SPLINE
SPL {X  -157.404, Y  +360.095, Z    +0.000, E1   +17.695, E3 +109849.442}
SPL {X  -159.413, Y  +375.108, Z    +0.000, E1    +9.284, E3 +109858.530}
SPL {X  -159.978, Y  +386.135, Z    +0.000, E1    +2.544, E3 +109862.092}
SPL {X  -160.000, Y  +393.708, Z    +0.000, E1    -3.216, E3 +109863.846}
SPL {X  -160.000, Y  +400.474, Z    +0.000, E1    -9.529, E3 +109865.892}
SPL {X  -160.000, Y  +409.652, Z    +0.000, E1   -18.026, E3 +109870.028}
SPL {X  -160.000, Y  +437.804, Z    +0.000, E1   -34.779, E3 +109894.821}
SPL {X  -160.000, Y  +463.067, Z    +0.000, E1   -38.672, E3 +109940.521}
SPL {X  -160.000, Y  +469.167, Z    +0.000, E1   -38.717, E3 +109956.627}
SPL {X  -160.000, Y  +476.691, Z    +0.000, E1   -38.728, E3 +109976.559}
SPL {X  -160.000, Y  +483.419, Z    +0.000, E1   -38.692, E3 +109994.459}
SPL {X  -160.000, Y  +489.013, Z    +0.000, E1   -38.683, E3 +110009.298}
SPL {X  -160.000, Y  +494.786, Z    +0.000, E1   -38.693, E3 +110024.608}
SPL {X  -160.000, Y  +500.108, Z    +0.000, E1   -38.668, E3 +110038.759}
SPL {X  -160.000, Y  +504.903, Z    +0.000, E1   -38.673, E3 +110051.480}
SPL {X  -160.000, Y  +510.180, Z    +0.000, E1   -38.675, E3 +110065.485}
SPL {X  -160.000, Y  +515.083, Z    +0.000, E1   -38.662, E3 +110078.505}
SPL {X  -160.000, Y  +520.479, Z    +0.000, E1   -38.692, E3 +110092.779}
SPL {X  -160.000, Y  +525.998, Z    +0.000, E1   -38.666, E3 +110107.457}
SPL {X  -160.000, Y  +531.341, Z    +0.000, E1   -38.684, E3 +110121.601}
SPL {X  -160.000, Y  +537.313, Z    +0.000, E1   -38.686, E3 +110137.441}
SPL {X  -160.000, Y  +543.203, Z    +0.000, E1   -38.679, E3 +110153.067}
SPL {X  -160.000, Y  +551.201, Z    +0.000, E1   -38.768, E3 +110174.128}
SPL {X  -160.000, Y  +561.335, Z    +0.000, E1   -38.777, E3 +110200.998}
SPL {X  -160.000, Y  +568.812, Z    +0.000, E1   -38.671, E3 +110221.001}
SPL {X  -160.000, Y  +574.116, Z    +0.000, E1   -38.680, E3 +110235.072}
SPL {X  -160.000, Y  +582.193, Z    +0.000, E1   -38.759, E3 +110256.375}
SPL {X  -160.000, Y  +591.932, Z    +0.000, E1   -38.763, E3 +110282.200}
SPL {X  -160.000, Y  +601.488, Z    +0.000, E1   -38.747, E3 +110307.576}
SPL {X  -160.000, Y  +609.161, Z    +0.000, E1   -38.685, E3 +110328.027}
SPL {X  -160.000, Y  +614.445, Z    +0.000, E1   -38.661, E3 +110342.077}
SPL {X  -160.000, Y  +621.895, Z    +0.000, E1   -38.769, E3 +110361.665}
SPL {X  -160.000, Y  +631.692, Z    +0.000, E1   -38.748, E3 +110387.718}
SPL {X  -160.000, Y  +639.246, Z    +0.000, E1   -38.671, E3 +110407.894}
SPL {X  -160.000, Y  +644.827, Z    +0.000, E1   -38.662, E3 +110422.728}
SPL {X  -160.000, Y  +650.491, Z    +0.000, E1   -38.673, E3 +110437.716}
SPL {X  -160.000, Y  +656.011, Z    +0.000, E1   -38.669, E3 +110452.369}
SPL {X  -160.000, Y  +661.156, Z    +0.000, E1   -38.659, E3 +110466.044}
SPL {X  -160.000, Y  +666.701, Z    +0.000, E1   -38.683, E3 +110480.704}
SPL {X  -159.961, Y  +675.011, Z    +0.000, E1   -38.755, E3 +110502.691}
SPL {X  -159.451, Y  +684.743, Z    +0.000, E1   -38.666, E3 +110529.044}
SPL {X  -158.386, Y  +694.170, Z    +0.000, E1   -38.484, E3 +110555.163}
SPL {X  -157.286, Y  +700.846, Z    +0.000, E1   -38.194, E3 +110574.130}
SPL {X  -156.328, Y  +705.580, Z    +0.000, E1   -38.037, E3 +110587.666}
SPL {X  -155.162, Y  +710.549, Z    +0.000, E1   -37.822, E3 +110602.070}
SPL {X  -153.914, Y  +715.210, Z    +0.000, E1   -37.596, E3 +110615.720}
SPL {X  -152.686, Y  +719.322, Z    +0.000, E1   -37.361, E3 +110627.892}
SPL {X  -150.251, Y  +726.496, Z    +0.000, E1   -33.848, E3 +110676.388}
ENDSPLINE

SPLINE
SPL {X  -156.089, Y  +706.662, Z    +0.000, E1   -21.279, E3 +110729.041}
SPL {X  -159.059, Y  +688.824, Z    +0.000, E1   -11.551, E3 +110743.002}
SPL {X  -159.959, Y  +675.119, Z    +0.000, E1    -3.373, E3 +110747.830}
SPL {X  -160.000, Y  +666.447, Z    +0.000, E1    +3.005, E3 +110749.864}
SPL {X  -160.000, Y  +658.774, Z    +0.000, E1   +10.317, E3 +110752.123}
SPL {X  -160.000, Y  +647.765, Z    +0.000, E1   +20.359, E3 +110757.488}
SPL {X  -160.000, Y  +622.607, Z    +0.000, E1   +34.692, E3 +110780.356}
SPL {X  -160.000, Y  +596.106, Z    +0.000, E1   +39.718, E3 +110822.356}
SPL {X  -160.000, Y  +592.273, Z    +0.000, E1   +39.746, E3 +110832.093}
SPL {X  -160.000, Y  +586.287, Z    +0.000, E1   +39.762, E3 +110847.352}
SPL {X  -160.000, Y  +577.753, Z    +0.000, E1   +39.844, E3 +110868.994}
SPL {X  -160.000, Y  +567.367, Z    +0.000, E1   +39.853, E3 +110895.488}
SPL {X  -160.000, Y  +559.466, Z    +0.000, E1   +39.761, E3 +110915.770}
SPL {X  -160.000, Y  +552.914, Z    +0.000, E1   +39.787, E3 +110932.437}
SPL {X  -160.000, Y  +546.390, Z    +0.000, E1   +39.760, E3 +110949.151}
SPL {X  -160.000, Y  +540.123, Z    +0.000, E1   +39.770, E3 +110965.130}
SPL {X  -160.000, Y  +533.658, Z    +0.000, E1   +39.771, E3 +110981.628}
SPL {X  -160.000, Y  +527.046, Z    +0.000, E1   +39.771, E3 +110998.504}
SPL {X  -160.000, Y  +521.063, Z    +0.000, E1   +39.756, E3 +111013.789}
SPL {X  -160.000, Y  +515.110, Z    +0.000, E1   +39.770, E3 +111028.961}
SPL {X  -160.000, Y  +508.717, Z    +0.000, E1   +39.766, E3 +111045.280}
SPL {X  -160.000, Y  +502.133, Z    +0.000, E1   +39.780, E3 +111062.046}
ENDSPLINE

SPLINE
SPL {X  -160.000, Y  +512.949, Z    +0.000, E1   +32.050, E3 +111078.304}
ENDSPLINE

SPLINE
SPL {X  -160.000, Y  +507.092, Z    +0.000, E1   +32.805, E3 +111092.932}
SPL {X  -160.000, Y  +499.824, Z    +0.000, E1   +34.003, E3 +111108.674}
SPL {X  -160.000, Y  +491.367, Z    +0.000, E1   +35.449, E3 +111125.414}
SPL {X  -160.000, Y  +483.082, Z    +0.000, E1   +36.782, E3 +111141.253}
SPL {X  -160.000, Y  +474.521, Z    +0.000, E1   +38.037, E3 +111157.341}
SPL {X  -160.000, Y  +465.343, Z    +0.000, E1   +38.802, E3 +111177.500}
SPL {X  -160.000, Y  +457.266, Z    +0.000, E1   +38.756, E3 +111198.953}
SPL {X  -160.000, Y  +448.553, Z    +0.000, E1   +38.823, E3 +111221.904}
SPL {X  -160.000, Y  +439.425, Z    +0.000, E1   +38.797, E3 +111246.075}
SPL {X  -160.000, Y  +430.351, Z    +0.000, E1   +38.810, E3 +111270.090}
SPL {X  -160.000, Y  +421.477, Z    +0.000, E1   +38.792, E3 +111293.594}
SPL {X  -160.000, Y  +412.292, Z    +0.000, E1   +38.825, E3 +111317.821}
SPL {X  -160.000, Y  +403.281, Z    +0.000, E1   +38.797, E3 +111341.701}
SPL {X  -160.000, Y  +394.948, Z    +0.000, E1   +38.796, E3 +111363.743}
SPL {X  -159.971, Y  +385.741, Z    +0.000, E1   +38.831, E3 +111388.064}
SPL {X  -159.525, Y  +376.478, Z    +0.000, E1   +38.739, E3 +111413.055}
SPL {X  -158.721, Y  +368.613, Z    +0.000, E1   +38.561, E3 +111434.778}
SPL {X  -157.505, Y  +360.654, Z    +0.000, E1   +38.390, E3 +111457.052}
SPL {X  -156.229, Y  +354.269, Z    +0.000, E1   +38.076, E3 +111475.401}
SPL {X  -155.202, Y  +349.910, Z    +0.000, E1   +37.893, E3 +111487.976}
SPL {X  -154.128, Y  +345.852, Z    +0.000, E1   +37.701, E3 +111499.800}
SPL {X  -152.890, Y  +341.633, Z    +0.000, E1   +37.487, E3 +111512.232}
SPL {X  -150.284, Y  +333.893, Z    +0.000, E1   +33.433, E3 +111567.042}
ENDSPLINE

SPLINE
SPL {X  -157.404, Y  +360.095, Z    +0.000, E1   +17.695, E3 +111622.167}
SPL {X  -159.413, Y  +375.108, Z    +0.000, E1    +9.284, E3 +111631.256}
SPL {X  -159.978, Y  +386.135, Z    +0.000, E1    +2.544, E3 +111634.817}
SPL {X  -160.000, Y  +393.708, Z    +0.000, E1    -3.216, E3 +111636.571}
SPL {X  -160.000, Y  +400.474, Z    +0.000, E1    -9.529, E3 +111638.617}
SPL {X  -160.000, Y  +409.652, Z    +0.000, E1   -18.026, E3 +111642.754}
SPL {X  -160.000, Y  +437.804, Z    +0.000, E1   -34.779, E3 +111667.546}
SPL {X  -160.000, Y  +463.067, Z    +0.000, E1   -38.672, E3 +111713.246}
SPL {X  -160.000, Y  +469.167, Z    +0.000, E1   -38.717, E3 +111729.353}
SPL {X  -160.000, Y  +476.691, Z    +0.000, E1   -38.728, E3 +111749.284}
SPL {X  -160.000, Y  +483.419, Z    +0.000, E1   -38.692, E3 +111767.185}
SPL {X  -160.000, Y  +489.013, Z    +0.000, E1   -38.683, E3 +111782.023}
SPL {X  -160.000, Y  +494.786, Z    +0.000, E1   -38.693, E3 +111797.333}
SPL {X  -160.000, Y  +500.108, Z    +0.000, E1   -38.668, E3 +111811.485}
SPL {X  -160.000, Y  +504.903, Z    +0.000, E1   -38.673, E3 +111824.206}
SPL {X  -160.000, Y  +510.180, Z    +0.000, E1   -38.675, E3 +111838.210}
SPL {X  -160.000, Y  +515.083, Z    +0.000, E1   -38.662, E3 +111851.230}
SPL {X  -160.000, Y  +520.479, Z    +0.000, E1   -38.692, E3 +111865.504}
SPL {X  -160.000, Y  +525.998, Z    +0.000, E1   -38.666, E3 +111880.182}
SPL {X  -160.000, Y  +531.341, Z    +0.000, E1   -38.684, E3 +111894.327}
SPL {X  -160.000, Y  +537.313, Z    +0.000, E1   -38.686, E3 +111910.166}
SPL {X  -160.000, Y  +543.203, Z    +0.000, E1   -38.679, E3 +111925.792}
SPL {X  -160.000, Y  +551.201, Z    +0.000, E1   -38.768, E3 +111946.853}
SPL {X  -160.000, Y  +561.335, Z    +0.000, E1   -38.777, E3 +111973.723}
SPL {X  -160.000, Y  +568.812, Z    +0.000, E1   -38.671, E3 +111993.727}
SPL {X  -160.000, Y  +574.116, Z    +0.000, E1   -38.680, E3 +112007.797}
SPL {X  -160.000, Y  +582.193, Z    +0.000, E1   -38.759, E3 +112029.101}
SPL {X  -160.000, Y  +591.932, Z    +0.000, E1   -38.763, E3 +112054.926}
SPL {X  -160.000, Y  +601.488, Z    +0.000, E1   -38.747, E3 +112080.301}
SPL {X  -160.000, Y  +609.161, Z    +0.000, E1   -38.685, E3 +112100.753}
SPL {X  -160.000, Y  +614.445, Z    +0.000, E1   -38.661, E3 +112114.802}
SPL {X  -160.000, Y  +621.895, Z    +0.000, E1   -38.769, E3 +112134.390}
SPL {X  -160.000, Y  +631.692, Z    +0.000, E1   -38.748, E3 +112160.443}
SPL {X  -160.000, Y  +639.246, Z    +0.000, E1   -38.671, E3 +112180.619}
SPL {X  -160.000, Y  +644.827, Z    +0.000, E1   -38.662, E3 +112195.454}
SPL {X  -160.000, Y  +650.491, Z    +0.000, E1   -38.673, E3 +112210.441}
SPL {X  -160.000, Y  +656.011, Z    +0.000, E1   -38.669, E3 +112225.094}
SPL {X  -160.000, Y  +661.156, Z    +0.000, E1   -38.659, E3 +112238.769}
SPL {X  -160.000, Y  +666.701, Z    +0.000, E1   -38.683, E3 +112253.429}
SPL {X  -159.961, Y  +675.011, Z    +0.000, E1   -38.755, E3 +112275.416}
SPL {X  -159.451, Y  +684.743, Z    +0.000, E1   -38.666, E3 +112301.769}
SPL {X  -158.386, Y  +694.170, Z    +0.000, E1   -38.484, E3 +112327.888}
SPL {X  -157.286, Y  +700.846, Z    +0.000, E1   -38.194, E3 +112346.856}
SPL {X  -156.328, Y  +705.580, Z    +0.000, E1   -38.037, E3 +112360.392}
SPL {X  -155.162, Y  +710.549, Z    +0.000, E1   -37.822, E3 +112374.796}
SPL {X  -153.914, Y  +715.210, Z    +0.000, E1   -37.596, E3 +112388.445}
SPL {X  -152.686, Y  +719.322, Z    +0.000, E1   -37.361, E3 +112400.617}
SPL {X  -150.251, Y  +726.496, Z    +0.000, E1   -33.848, E3 +112449.113}
ENDSPLINE

SPLINE
SPL {X  -156.089, Y  +706.662, Z    +0.000, E1   -21.279, E3 +112501.766}
SPL {X  -159.059, Y  +688.824, Z    +0.000, E1   -11.551, E3 +112515.727}
SPL {X  -159.959, Y  +675.119, Z    +0.000, E1    -3.373, E3 +112520.555}
SPL {X  -160.000, Y  +666.447, Z    +0.000, E1    +3.005, E3 +112522.590}
SPL {X  -160.000, Y  +658.774, Z    +0.000, E1   +10.317, E3 +112524.848}
SPL {X  -160.000, Y  +647.765, Z    +0.000, E1   +20.359, E3 +112530.213}
SPL {X  -160.000, Y  +622.607, Z    +0.000, E1   +34.692, E3 +112553.081}
SPL {X  -160.000, Y  +593.120, Z    +0.000, E1   +39.775, E3 +112602.611}
SPL {X  -160.000, Y  +586.287, Z    +0.000, E1   +39.762, E3 +112620.078}
SPL {X  -160.000, Y  +577.753, Z    +0.000, E1   +39.844, E3 +112641.719}
SPL {X  -160.000, Y  +567.367, Z    +0.000, E1   +39.853, E3 +112668.213}
SPL {X  -160.000, Y  +559.466, Z    +0.000, E1   +39.761, E3 +112688.495}
SPL {X  -160.000, Y  +552.914, Z    +0.000, E1   +39.787, E3 +112705.162}
SPL {X  -160.000, Y  +546.390, Z    +0.000, E1   +39.760, E3 +112721.876}
SPL {X  -160.000, Y  +540.123, Z    +0.000, E1   +39.770, E3 +112737.855}
SPL {X  -160.000, Y  +533.658, Z    +0.000, E1   +39.771, E3 +112754.354}
SPL {X  -160.000, Y  +527.046, Z    +0.000, E1   +39.771, E3 +112771.230}
SPL {X  -160.000, Y  +521.063, Z    +0.000, E1   +39.756, E3 +112786.514}
SPL {X  -160.000, Y  +515.110, Z    +0.000, E1   +39.770, E3 +112801.687}
SPL {X  -160.000, Y  +508.717, Z    +0.000, E1   +39.766, E3 +112818.005}
SPL {X  -160.000, Y  +502.133, Z    +0.000, E1   +39.780, E3 +112834.771}
ENDSPLINE

SPLINE
SPL {X  -160.000, Y  +512.949, Z    +0.000, E1   +32.050, E3 +112851.029}
ENDSPLINE

SPLINE
SPL {X  -160.000, Y  +507.092, Z    +0.000, E1   +32.805, E3 +112865.657}
SPL {X  -160.000, Y  +499.824, Z    +0.000, E1   +34.003, E3 +112881.399}
SPL {X  -160.000, Y  +491.367, Z    +0.000, E1   +35.449, E3 +112898.139}
SPL {X  -160.000, Y  +483.082, Z    +0.000, E1   +36.782, E3 +112913.978}
SPL {X  -160.000, Y  +474.521, Z    +0.000, E1   +38.037, E3 +112930.066}
SPL {X  -160.000, Y  +465.343, Z    +0.000, E1   +38.802, E3 +112950.225}
SPL {X  -160.000, Y  +457.266, Z    +0.000, E1   +38.756, E3 +112971.679}
SPL {X  -160.000, Y  +448.553, Z    +0.000, E1   +38.823, E3 +112994.630}
SPL {X  -160.000, Y  +439.425, Z    +0.000, E1   +38.797, E3 +113018.801}
SPL {X  -160.000, Y  +430.351, Z    +0.000, E1   +38.810, E3 +113042.815}
SPL {X  -160.000, Y  +421.477, Z    +0.000, E1   +38.792, E3 +113066.319}
SPL {X  -160.000, Y  +412.292, Z    +0.000, E1   +38.825, E3 +113090.547}
SPL {X  -160.000, Y  +403.281, Z    +0.000, E1   +38.797, E3 +113114.426}
SPL {X  -160.000, Y  +394.948, Z    +0.000, E1   +38.796, E3 +113136.468}
SPL {X  -159.971, Y  +385.741, Z    +0.000, E1   +38.831, E3 +113160.789}
SPL {X  -159.525, Y  +376.478, Z    +0.000, E1   +38.739, E3 +113185.780}
SPL {X  -158.721, Y  +368.613, Z    +0.000, E1   +38.561, E3 +113207.504}
SPL {X  -157.505, Y  +360.654, Z    +0.000, E1   +38.390, E3 +113229.777}
SPL {X  -156.229, Y  +354.269, Z    +0.000, E1   +38.076, E3 +113248.126}
SPL {X  -155.202, Y  +349.910, Z    +0.000, E1   +37.893, E3 +113260.701}
SPL {X  -154.128, Y  +345.852, Z    +0.000, E1   +37.701, E3 +113272.525}
SPL {X  -152.890, Y  +341.633, Z    +0.000, E1   +37.487, E3 +113284.957}
SPL {X  -150.284, Y  +333.893, Z    +0.000, E1   +33.433, E3 +113339.767}
ENDSPLINE

SPLINE
SPL {X  -157.404, Y  +360.095, Z    +0.000, E1   +17.695, E3 +113394.892}
SPL {X  -159.413, Y  +375.108, Z    +0.000, E1    +9.284, E3 +113403.981}
SPL {X  -159.978, Y  +386.135, Z    +0.000, E1    +2.544, E3 +113407.542}
SPL {X  -160.000, Y  +393.708, Z    +0.000, E1    -3.216, E3 +113409.296}
SPL {X  -160.000, Y  +400.474, Z    +0.000, E1    -9.529, E3 +113411.342}
SPL {X  -160.000, Y  +409.652, Z    +0.000, E1   -18.026, E3 +113415.479}
SPL {X  -160.000, Y  +437.804, Z    +0.000, E1   -34.779, E3 +113440.272}
SPL {X  -160.000, Y  +463.067, Z    +0.000, E1   -38.672, E3 +113485.972}
SPL {X  -160.000, Y  +469.167, Z    +0.000, E1   -38.717, E3 +113502.078}
SPL {X  -160.000, Y  +476.691, Z    +0.000, E1   -38.728, E3 +113522.009}
SPL {X  -160.000, Y  +483.419, Z    +0.000, E1   -38.692, E3 +113539.910}
SPL {X  -160.000, Y  +489.013, Z    +0.000, E1   -38.683, E3 +113554.748}
SPL {X  -160.000, Y  +494.786, Z    +0.000, E1   -38.693, E3 +113570.058}
SPL {X  -160.000, Y  +500.108, Z    +0.000, E1   -38.668, E3 +113584.210}
SPL {X  -160.000, Y  +504.903, Z    +0.000, E1   -38.673, E3 +113596.931}
SPL {X  -160.000, Y  +510.180, Z    +0.000, E1   -38.675, E3 +113610.935}
SPL {X  -160.000, Y  +515.083, Z    +0.000, E1   -38.662, E3 +113623.955}
SPL {X  -160.000, Y  +520.479, Z    +0.000, E1   -38.692, E3 +113638.229}
SPL {X  -160.000, Y  +525.998, Z    +0.000, E1   -38.666, E3 +113652.908}
SPL {X  -160.000, Y  +531.341, Z    +0.000, E1   -38.684, E3 +113667.052}
SPL {X  -160.000, Y  +537.313, Z    +0.000, E1   -38.686, E3 +113682.892}
SPL {X  -160.000, Y  +543.203, Z    +0.000, E1   -38.679, E3 +113698.517}
SPL {X  -160.000, Y  +551.201, Z    +0.000, E1   -38.768, E3 +113719.578}
SPL {X  -160.000, Y  +561.335, Z    +0.000, E1   -38.777, E3 +113746.449}
SPL {X  -160.000, Y  +568.812, Z    +0.000, E1   -38.671, E3 +113766.452}
SPL {X  -160.000, Y  +574.116, Z    +0.000, E1   -38.680, E3 +113780.522}
SPL {X  -160.000, Y  +582.193, Z    +0.000, E1   -38.759, E3 +113801.826}
SPL {X  -160.000, Y  +591.932, Z    +0.000, E1   -38.763, E3 +113827.651}
SPL {X  -160.000, Y  +601.488, Z    +0.000, E1   -38.747, E3 +113853.026}
SPL {X  -160.000, Y  +609.161, Z    +0.000, E1   -38.685, E3 +113873.478}
SPL {X  -160.000, Y  +614.445, Z    +0.000, E1   -38.661, E3 +113887.527}
SPL {X  -160.000, Y  +621.895, Z    +0.000, E1   -38.769, E3 +113907.115}
SPL {X  -160.000, Y  +631.692, Z    +0.000, E1   -38.748, E3 +113933.169}
SPL {X  -160.000, Y  +639.246, Z    +0.000, E1   -38.671, E3 +113953.344}
SPL {X  -160.000, Y  +644.827, Z    +0.000, E1   -38.662, E3 +113968.179}
SPL {X  -160.000, Y  +650.491, Z    +0.000, E1   -38.673, E3 +113983.166}
SPL {X  -160.000, Y  +656.011, Z    +0.000, E1   -38.669, E3 +113997.819}
SPL {X  -160.000, Y  +661.156, Z    +0.000, E1   -38.659, E3 +114011.494}
SPL {X  -160.000, Y  +666.701, Z    +0.000, E1   -38.683, E3 +114026.155}
SPL {X  -159.961, Y  +675.011, Z    +0.000, E1   -38.755, E3 +114048.141}
SPL {X  -159.451, Y  +684.743, Z    +0.000, E1   -38.666, E3 +114074.495}
SPL {X  -158.386, Y  +694.170, Z    +0.000, E1   -38.484, E3 +114100.613}
SPL {X  -157.286, Y  +700.846, Z    +0.000, E1   -38.194, E3 +114119.581}
SPL {X  -156.328, Y  +705.580, Z    +0.000, E1   -38.037, E3 +114133.117}
SPL {X  -155.162, Y  +710.549, Z    +0.000, E1   -37.822, E3 +114147.521}
SPL {X  -153.914, Y  +715.210, Z    +0.000, E1   -37.596, E3 +114161.170}
SPL {X  -152.686, Y  +719.322, Z    +0.000, E1   -37.361, E3 +114173.342}
SPL {X  -150.251, Y  +726.496, Z    +0.000, E1   -33.848, E3 +114221.838}
ENDSPLINE

SPLINE
SPL {X  -156.089, Y  +706.662, Z    +0.000, E1   -21.279, E3 +114274.491}
SPL {X  -159.059, Y  +688.824, Z    +0.000, E1   -11.551, E3 +114288.452}
SPL {X  -159.959, Y  +675.119, Z    +0.000, E1    -3.373, E3 +114293.280}
SPL {X  -160.000, Y  +666.447, Z    +0.000, E1    +3.005, E3 +114295.315}
SPL {X  -160.000, Y  +658.774, Z    +0.000, E1   +10.317, E3 +114297.574}
SPL {X  -160.000, Y  +647.765, Z    +0.000, E1   +20.359, E3 +114302.939}
SPL {X  -160.000, Y  +622.607, Z    +0.000, E1   +34.692, E3 +114325.806}
SPL {X  -160.000, Y  +596.106, Z    +0.000, E1   +39.718, E3 +114367.806}
SPL {X  -160.000, Y  +592.273, Z    +0.000, E1   +39.746, E3 +114377.543}
SPL {X  -160.000, Y  +586.287, Z    +0.000, E1   +39.762, E3 +114392.803}
SPL {X  -160.000, Y  +577.753, Z    +0.000, E1   +39.844, E3 +114414.444}
SPL {X  -160.000, Y  +567.367, Z    +0.000, E1   +39.853, E3 +114440.939}
SPL {X  -160.000, Y  +559.466, Z    +0.000, E1   +39.761, E3 +114461.220}
SPL {X  -160.000, Y  +552.914, Z    +0.000, E1   +39.787, E3 +114477.887}
SPL {X  -160.000, Y  +546.390, Z    +0.000, E1   +39.760, E3 +114494.601}
SPL {X  -160.000, Y  +540.123, Z    +0.000, E1   +39.770, E3 +114510.580}
SPL {X  -160.000, Y  +533.658, Z    +0.000, E1   +39.771, E3 +114527.079}
SPL {X  -160.000, Y  +527.046, Z    +0.000, E1   +39.771, E3 +114543.955}
SPL {X  -160.000, Y  +521.063, Z    +0.000, E1   +39.756, E3 +114559.239}
SPL {X  -160.000, Y  +515.110, Z    +0.000, E1   +39.770, E3 +114574.412}
SPL {X  -160.000, Y  +508.717, Z    +0.000, E1   +39.766, E3 +114590.730}
SPL {X  -160.000, Y  +502.133, Z    +0.000, E1   +39.780, E3 +114607.497}
ENDSPLINE

SPLINE
SPL {X  -160.000, Y  +512.949, Z    +0.000, E1   +32.050, E3 +114623.754}
ENDSPLINE

SPLINE
SPL {X  -160.000, Y  +507.092, Z    +0.000, E1   +32.805, E3 +114638.382}
SPL {X  -160.000, Y  +499.824, Z    +0.000, E1   +34.003, E3 +114654.124}
SPL {X  -160.000, Y  +491.367, Z    +0.000, E1   +35.449, E3 +114670.865}
SPL {X  -160.000, Y  +483.082, Z    +0.000, E1   +36.782, E3 +114686.703}
SPL {X  -160.000, Y  +474.521, Z    +0.000, E1   +38.037, E3 +114702.791}
SPL {X  -160.000, Y  +465.343, Z    +0.000, E1   +38.802, E3 +114722.950}
SPL {X  -160.000, Y  +457.266, Z    +0.000, E1   +38.756, E3 +114744.404}
SPL {X  -160.000, Y  +448.553, Z    +0.000, E1   +38.823, E3 +114767.355}
SPL {X  -160.000, Y  +439.425, Z    +0.000, E1   +38.797, E3 +114791.526}
SPL {X  -160.000, Y  +430.351, Z    +0.000, E1   +38.810, E3 +114815.541}
SPL {X  -160.000, Y  +421.477, Z    +0.000, E1   +38.792, E3 +114839.044}
SPL {X  -160.000, Y  +412.292, Z    +0.000, E1   +38.825, E3 +114863.272}
SPL {X  -160.000, Y  +403.281, Z    +0.000, E1   +38.797, E3 +114887.152}
SPL {X  -160.000, Y  +394.948, Z    +0.000, E1   +38.796, E3 +114909.193}
SPL {X  -159.971, Y  +385.741, Z    +0.000, E1   +38.831, E3 +114933.515}
SPL {X  -159.525, Y  +376.478, Z    +0.000, E1   +38.739, E3 +114958.506}
SPL {X  -158.721, Y  +368.613, Z    +0.000, E1   +38.561, E3 +114980.229}
SPL {X  -157.505, Y  +360.654, Z    +0.000, E1   +38.390, E3 +115002.502}
SPL {X  -156.229, Y  +354.269, Z    +0.000, E1   +38.076, E3 +115020.852}
SPL {X  -155.202, Y  +349.910, Z    +0.000, E1   +37.893, E3 +115033.426}
SPL {X  -154.128, Y  +345.852, Z    +0.000, E1   +37.701, E3 +115045.250}
SPL {X  -152.890, Y  +341.633, Z    +0.000, E1   +37.487, E3 +115057.682}
SPL {X  -150.284, Y  +333.893, Z    +0.000, E1   +33.433, E3 +115112.493}
ENDSPLINE

SPLINE
SPL {X  -157.404, Y  +360.095, Z    +0.000, E1   +17.695, E3 +115167.617}
SPL {X  -159.413, Y  +375.108, Z    +0.000, E1    +9.284, E3 +115176.706}
SPL {X  -159.978, Y  +386.135, Z    +0.000, E1    +2.544, E3 +115180.267}
SPL {X  -160.000, Y  +393.708, Z    +0.000, E1    -3.216, E3 +115182.021}
SPL {X  -160.000, Y  +400.474, Z    +0.000, E1    -9.529, E3 +115184.068}
SPL {X  -160.000, Y  +409.652, Z    +0.000, E1   -18.026, E3 +115188.204}
SPL {X  -160.000, Y  +437.804, Z    +0.000, E1   -34.779, E3 +115212.997}
SPL {X  -160.000, Y  +463.067, Z    +0.000, E1   -38.672, E3 +115258.697}
SPL {X  -160.000, Y  +469.167, Z    +0.000, E1   -38.717, E3 +115274.803}
SPL {X  -160.000, Y  +476.691, Z    +0.000, E1   -38.728, E3 +115294.735}
SPL {X  -160.000, Y  +483.419, Z    +0.000, E1   -38.692, E3 +115312.635}
SPL {X  -160.000, Y  +489.013, Z    +0.000, E1   -38.683, E3 +115327.474}
SPL {X  -160.000, Y  +494.786, Z    +0.000, E1   -38.693, E3 +115342.784}
SPL {X  -160.000, Y  +500.108, Z    +0.000, E1   -38.668, E3 +115356.935}
SPL {X  -160.000, Y  +504.903, Z    +0.000, E1   -38.673, E3 +115369.656}
SPL {X  -160.000, Y  +510.180, Z    +0.000, E1   -38.675, E3 +115383.661}
SPL {X  -160.000, Y  +515.083, Z    +0.000, E1   -38.662, E3 +115396.680}
SPL {X  -160.000, Y  +520.479, Z    +0.000, E1   -38.692, E3 +115410.955}
SPL {X  -160.000, Y  +525.998, Z    +0.000, E1   -38.666, E3 +115425.633}
SPL {X  -160.000, Y  +531.341, Z    +0.000, E1   -38.684, E3 +115439.777}
SPL {X  -160.000, Y  +537.313, Z    +0.000, E1   -38.686, E3 +115455.617}
SPL {X  -160.000, Y  +543.203, Z    +0.000, E1   -38.679, E3 +115471.242}
SPL {X  -160.000, Y  +551.201, Z    +0.000, E1   -38.768, E3 +115492.304}
SPL {X  -160.000, Y  +561.335, Z    +0.000, E1   -38.777, E3 +115519.174}
SPL {X  -160.000, Y  +568.812, Z    +0.000, E1   -38.671, E3 +115539.177}
SPL {X  -160.000, Y  +574.116, Z    +0.000, E1   -38.680, E3 +115553.248}
SPL {X  -160.000, Y  +582.193, Z    +0.000, E1   -38.759, E3 +115574.551}
SPL {X  -160.000, Y  +591.932, Z    +0.000, E1   -38.763, E3 +115600.376}
SPL {X  -160.000, Y  +601.488, Z    +0.000, E1   -38.747, E3 +115625.751}
SPL {X  -160.000, Y  +609.161, Z    +0.000, E1   -38.685, E3 +115646.203}
SPL {X  -160.000, Y  +614.445, Z    +0.000, E1   -38.661, E3 +115660.252}
SPL {X  -160.000, Y  +621.895, Z    +0.000, E1   -38.769, E3 +115679.840}
SPL {X  -160.000, Y  +631.692, Z    +0.000, E1   -38.748, E3 +115705.894}
SPL {X  -160.000, Y  +639.246, Z    +0.000, E1   -38.671, E3 +115726.069}
SPL {X  -160.000, Y  +644.827, Z    +0.000, E1   -38.662, E3 +115740.904}
SPL {X  -160.000, Y  +650.491, Z    +0.000, E1   -38.673, E3 +115755.892}
SPL {X  -160.000, Y  +656.011, Z    +0.000, E1   -38.669, E3 +115770.545}
SPL {X  -160.000, Y  +661.156, Z    +0.000, E1   -38.659, E3 +115784.220}
SPL {X  -160.000, Y  +666.701, Z    +0.000, E1   -38.683, E3 +115798.880}
SPL {X  -159.961, Y  +675.011, Z    +0.000, E1   -38.755, E3 +115820.866}
SPL {X  -159.451, Y  +684.743, Z    +0.000, E1   -38.666, E3 +115847.220}
SPL {X  -158.386, Y  +694.170, Z    +0.000, E1   -38.484, E3 +115873.338}
SPL {X  -157.286, Y  +700.846, Z    +0.000, E1   -38.194, E3 +115892.306}
SPL {X  -156.328, Y  +705.580, Z    +0.000, E1   -38.037, E3 +115905.842}
SPL {X  -155.162, Y  +710.549, Z    +0.000, E1   -37.822, E3 +115920.246}
SPL {X  -153.914, Y  +715.210, Z    +0.000, E1   -37.596, E3 +115933.895}
SPL {X  -152.686, Y  +719.322, Z    +0.000, E1   -37.361, E3 +115946.068}
SPL {X  -150.251, Y  +726.496, Z    +0.000, E1   -33.848, E3 +115994.563}
ENDSPLINE

SPLINE
SPL {X  -156.089, Y  +706.662, Z    +0.000, E1   -21.279, E3 +116047.217}
SPL {X  -159.059, Y  +688.824, Z    +0.000, E1   -11.551, E3 +116061.177}
SPL {X  -159.959, Y  +675.119, Z    +0.000, E1    -3.373, E3 +116066.005}
SPL {X  -160.000, Y  +666.447, Z    +0.000, E1    +3.005, E3 +116068.040}
SPL {X  -160.000, Y  +658.774, Z    +0.000, E1   +10.317, E3 +116070.299}
SPL {X  -160.000, Y  +647.765, Z    +0.000, E1   +20.359, E3 +116075.664}
SPL {X  -160.000, Y  +622.607, Z    +0.000, E1   +34.692, E3 +116098.531}
SPL {X  -160.000, Y  +593.120, Z    +0.000, E1   +39.775, E3 +116148.061}
SPL {X  -160.000, Y  +586.287, Z    +0.000, E1   +39.762, E3 +116165.528}
SPL {X  -160.000, Y  +577.753, Z    +0.000, E1   +39.844, E3 +116187.170}
SPL {X  -160.000, Y  +567.367, Z    +0.000, E1   +39.853, E3 +116213.664}
SPL {X  -160.000, Y  +559.466, Z    +0.000, E1   +39.761, E3 +116233.945}
SPL {X  -160.000, Y  +552.914, Z    +0.000, E1   +39.787, E3 +116250.613}
SPL {X  -160.000, Y  +546.390, Z    +0.000, E1   +39.760, E3 +116267.326}
SPL {X  -160.000, Y  +540.123, Z    +0.000, E1   +39.770, E3 +116283.306}
SPL {X  -160.000, Y  +533.658, Z    +0.000, E1   +39.771, E3 +116299.804}
SPL {X  -160.000, Y  +527.046, Z    +0.000, E1   +39.771, E3 +116316.680}
SPL {X  -160.000, Y  +521.063, Z    +0.000, E1   +39.756, E3 +116331.965}
SPL {X  -160.000, Y  +515.110, Z    +0.000, E1   +39.770, E3 +116347.137}
SPL {X  -160.000, Y  +508.717, Z    +0.000, E1   +39.766, E3 +116363.455}
SPL {X  -160.000, Y  +502.133, Z    +0.000, E1   +39.780, E3 +116380.222}
ENDSPLINE

SPLINE
SPL {X  -160.000, Y  +512.949, Z    +0.000, E1   +32.050, E3 +116396.479}
ENDSPLINE

SPLINE
SPL {X  -160.000, Y  +507.092, Z    +0.000, E1   +32.805, E3 +116411.108}
SPL {X  -160.000, Y  +499.824, Z    +0.000, E1   +34.003, E3 +116426.849}
SPL {X  -160.000, Y  +491.367, Z    +0.000, E1   +35.449, E3 +116443.590}
SPL {X  -160.000, Y  +483.082, Z    +0.000, E1   +36.782, E3 +116459.429}
SPL {X  -160.000, Y  +474.521, Z    +0.000, E1   +38.037, E3 +116475.517}
SPL {X  -160.000, Y  +465.343, Z    +0.000, E1   +38.802, E3 +116495.675}
SPL {X  -160.000, Y  +457.266, Z    +0.000, E1   +38.756, E3 +116517.129}
SPL {X  -160.000, Y  +448.553, Z    +0.000, E1   +38.823, E3 +116540.080}
SPL {X  -160.000, Y  +439.425, Z    +0.000, E1   +38.797, E3 +116564.251}
SPL {X  -160.000, Y  +430.351, Z    +0.000, E1   +38.810, E3 +116588.266}
SPL {X  -160.000, Y  +421.477, Z    +0.000, E1   +38.792, E3 +116611.770}
SPL {X  -160.000, Y  +412.292, Z    +0.000, E1   +38.825, E3 +116635.997}
SPL {X  -160.000, Y  +403.281, Z    +0.000, E1   +38.797, E3 +116659.877}
SPL {X  -160.000, Y  +394.948, Z    +0.000, E1   +38.796, E3 +116681.919}
SPL {X  -159.971, Y  +385.741, Z    +0.000, E1   +38.831, E3 +116706.240}
SPL {X  -159.525, Y  +376.478, Z    +0.000, E1   +38.739, E3 +116731.231}
SPL {X  -158.721, Y  +368.613, Z    +0.000, E1   +38.561, E3 +116752.954}
SPL {X  -157.505, Y  +360.654, Z    +0.000, E1   +38.390, E3 +116775.227}
SPL {X  -156.229, Y  +354.269, Z    +0.000, E1   +38.076, E3 +116793.577}
SPL {X  -155.202, Y  +349.910, Z    +0.000, E1   +37.893, E3 +116806.151}
SPL {X  -154.128, Y  +345.852, Z    +0.000, E1   +37.701, E3 +116817.975}
SPL {X  -152.890, Y  +341.633, Z    +0.000, E1   +37.487, E3 +116830.407}
SPL {X  -150.284, Y  +333.893, Z    +0.000, E1   +33.433, E3 +116885.218}
ENDSPLINE

SPLINE
SPL {X  -157.404, Y  +360.095, Z    +0.000, E1   +17.695, E3 +116940.343}
SPL {X  -159.413, Y  +375.108, Z    +0.000, E1    +9.284, E3 +116949.431}
SPL {X  -159.978, Y  +386.135, Z    +0.000, E1    +2.544, E3 +116952.993}
SPL {X  -160.000, Y  +393.708, Z    +0.000, E1    -3.216, E3 +116954.746}
SPL {X  -160.000, Y  +400.474, Z    +0.000, E1    -9.529, E3 +116956.793}
SPL {X  -160.000, Y  +409.652, Z    +0.000, E1   -18.026, E3 +116960.929}
SPL {X  -160.000, Y  +437.804, Z    +0.000, E1   -34.779, E3 +116985.722}
SPL {X  -160.000, Y  +463.067, Z    +0.000, E1   -38.672, E3 +117031.422}
SPL {X  -160.000, Y  +469.167, Z    +0.000, E1   -38.717, E3 +117047.528}
SPL {X  -160.000, Y  +476.691, Z    +0.000, E1   -38.728, E3 +117067.460}
SPL {X  -160.000, Y  +483.419, Z    +0.000, E1   -38.692, E3 +117085.360}
SPL {X  -160.000, Y  +489.013, Z    +0.000, E1   -38.683, E3 +117100.199}
SPL {X  -160.000, Y  +494.786, Z    +0.000, E1   -38.693, E3 +117115.509}
SPL {X  -160.000, Y  +500.108, Z    +0.000, E1   -38.668, E3 +117129.660}
SPL {X  -160.000, Y  +504.903, Z    +0.000, E1   -38.673, E3 +117142.381}
SPL {X  -160.000, Y  +510.180, Z    +0.000, E1   -38.675, E3 +117156.386}
SPL {X  -160.000, Y  +515.083, Z    +0.000, E1   -38.662, E3 +117169.405}
SPL {X  -160.000, Y  +520.479, Z    +0.000, E1   -38.692, E3 +117183.680}
SPL {X  -160.000, Y  +525.998, Z    +0.000, E1   -38.666, E3 +117198.358}
SPL {X  -160.000, Y  +531.341, Z    +0.000, E1   -38.684, E3 +117212.502}
SPL {X  -160.000, Y  +537.313, Z    +0.000, E1   -38.686, E3 +117228.342}
SPL {X  -160.000, Y  +543.203, Z    +0.000, E1   -38.679, E3 +117243.968}
SPL {X  -160.000, Y  +551.201, Z    +0.000, E1   -38.768, E3 +117265.029}
SPL {X  -160.000, Y  +561.335, Z    +0.000, E1   -38.777, E3 +117291.899}
SPL {X  -160.000, Y  +568.812, Z    +0.000, E1   -38.671, E3 +117311.902}
SPL {X  -160.000, Y  +574.116, Z    +0.000, E1   -38.680, E3 +117325.973}
SPL {X  -160.000, Y  +582.193, Z    +0.000, E1   -38.759, E3 +117347.276}
SPL {X  -160.000, Y  +591.932, Z    +0.000, E1   -38.763, E3 +117373.101}
SPL {X  -160.000, Y  +601.488, Z    +0.000, E1   -38.747, E3 +117398.477}
SPL {X  -160.000, Y  +609.161, Z    +0.000, E1   -38.685, E3 +117418.928}
SPL {X  -160.000, Y  +614.445, Z    +0.000, E1   -38.661, E3 +117432.978}
SPL {X  -160.000, Y  +621.895, Z    +0.000, E1   -38.769, E3 +117452.566}
SPL {X  -160.000, Y  +631.692, Z    +0.000, E1   -38.748, E3 +117478.619}
SPL {X  -160.000, Y  +639.246, Z    +0.000, E1   -38.671, E3 +117498.795}
SPL {X  -160.000, Y  +644.827, Z    +0.000, E1   -38.662, E3 +117513.629}
SPL {X  -160.000, Y  +650.491, Z    +0.000, E1   -38.673, E3 +117528.617}
SPL {X  -160.000, Y  +656.011, Z    +0.000, E1   -38.669, E3 +117543.270}
SPL {X  -160.000, Y  +661.156, Z    +0.000, E1   -38.659, E3 +117556.945}
SPL {X  -160.000, Y  +666.701, Z    +0.000, E1   -38.683, E3 +117571.605}
SPL {X  -159.961, Y  +675.011, Z    +0.000, E1   -38.755, E3 +117593.592}
SPL {X  -159.451, Y  +684.743, Z    +0.000, E1   -38.666, E3 +117619.945}
SPL {X  -158.386, Y  +694.170, Z    +0.000, E1   -38.484, E3 +117646.064}
SPL {X  -157.286, Y  +700.846, Z    +0.000, E1   -38.194, E3 +117665.031}
SPL {X  -156.328, Y  +705.580, Z    +0.000, E1   -38.037, E3 +117678.567}
SPL {X  -155.162, Y  +710.549, Z    +0.000, E1   -37.822, E3 +117692.971}
SPL {X  -153.914, Y  +715.210, Z    +0.000, E1   -37.596, E3 +117706.621}
SPL {X  -152.686, Y  +719.322, Z    +0.000, E1   -37.361, E3 +117718.793}
SPL {X  -150.251, Y  +726.496, Z    +0.000, E1   -33.848, E3 +117767.289}
ENDSPLINE

SPLINE
SPL {X  -156.089, Y  +706.662, Z    +0.000, E1   -21.279, E3 +117819.942}
SPL {X  -159.059, Y  +688.824, Z    +0.000, E1   -11.551, E3 +117833.902}
SPL {X  -159.959, Y  +675.119, Z    +0.000, E1    -3.373, E3 +117838.731}
SPL {X  -160.000, Y  +666.447, Z    +0.000, E1    +3.005, E3 +117840.765}
SPL {X  -160.000, Y  +658.774, Z    +0.000, E1   +10.317, E3 +117843.024}
SPL {X  -160.000, Y  +647.765, Z    +0.000, E1   +20.359, E3 +117848.389}
SPL {X  -160.000, Y  +622.607, Z    +0.000, E1   +34.692, E3 +117871.257}
SPL {X  -160.000, Y  +596.106, Z    +0.000, E1   +39.718, E3 +117913.256}
SPL {X  -160.000, Y  +592.273, Z    +0.000, E1   +39.746, E3 +117922.994}
SPL {X  -160.000, Y  +586.287, Z    +0.000, E1   +39.762, E3 +117938.253}
SPL {X  -160.000, Y  +577.753, Z    +0.000, E1   +39.844, E3 +117959.895}
SPL {X  -160.000, Y  +567.367, Z    +0.000, E1   +39.853, E3 +117986.389}
SPL {X  -160.000, Y  +559.466, Z    +0.000, E1   +39.761, E3 +118006.671}
SPL {X  -160.000, Y  +552.914, Z    +0.000, E1   +39.787, E3 +118023.338}
SPL {X  -160.000, Y  +546.390, Z    +0.000, E1   +39.760, E3 +118040.052}
SPL {X  -160.000, Y  +540.123, Z    +0.000, E1   +39.770, E3 +118056.031}
SPL {X  -160.000, Y  +533.658, Z    +0.000, E1   +39.771, E3 +118072.529}
SPL {X  -160.000, Y  +527.046, Z    +0.000, E1   +39.771, E3 +118089.405}
SPL {X  -160.000, Y  +521.063, Z    +0.000, E1   +39.756, E3 +118104.690}
SPL {X  -160.000, Y  +515.110, Z    +0.000, E1   +39.770, E3 +118119.862}
SPL {X  -160.000, Y  +508.717, Z    +0.000, E1   +39.766, E3 +118136.181}
SPL {X  -160.000, Y  +502.133, Z    +0.000, E1   +39.780, E3 +118152.947}
ENDSPLINE

SPLINE
SPL {X  -160.000, Y  +512.949, Z    +0.000, E1   +32.050, E3 +118169.204}
ENDSPLINE

SPLINE
SPL {X  -160.000, Y  +507.092, Z    +0.000, E1   +32.805, E3 +118183.833}
SPL {X  -160.000, Y  +499.824, Z    +0.000, E1   +34.003, E3 +118199.575}
SPL {X  -160.000, Y  +491.367, Z    +0.000, E1   +35.449, E3 +118216.315}
SPL {X  -160.000, Y  +483.082, Z    +0.000, E1   +36.782, E3 +118232.154}
SPL {X  -160.000, Y  +474.521, Z    +0.000, E1   +38.037, E3 +118248.242}
SPL {X  -160.000, Y  +465.343, Z    +0.000, E1   +38.802, E3 +118268.401}
SPL {X  -160.000, Y  +457.266, Z    +0.000, E1   +38.756, E3 +118289.854}
SPL {X  -160.000, Y  +448.553, Z    +0.000, E1   +38.823, E3 +118312.805}
SPL {X  -160.000, Y  +439.425, Z    +0.000, E1   +38.797, E3 +118336.976}
SPL {X  -160.000, Y  +430.351, Z    +0.000, E1   +38.810, E3 +118360.991}
SPL {X  -160.000, Y  +421.477, Z    +0.000, E1   +38.792, E3 +118384.495}
SPL {X  -160.000, Y  +412.292, Z    +0.000, E1   +38.825, E3 +118408.722}
SPL {X  -160.000, Y  +403.281, Z    +0.000, E1   +38.797, E3 +118432.602}
SPL {X  -160.000, Y  +394.948, Z    +0.000, E1   +38.796, E3 +118454.644}
SPL {X  -159.971, Y  +385.741, Z    +0.000, E1   +38.831, E3 +118478.965}
SPL {X  -159.525, Y  +376.478, Z    +0.000, E1   +38.739, E3 +118503.956}
SPL {X  -158.721, Y  +368.613, Z    +0.000, E1   +38.561, E3 +118525.679}
SPL {X  -157.505, Y  +360.654, Z    +0.000, E1   +38.390, E3 +118547.952}
SPL {X  -156.229, Y  +354.269, Z    +0.000, E1   +38.076, E3 +118566.302}
SPL {X  -155.202, Y  +349.910, Z    +0.000, E1   +37.893, E3 +118578.877}
SPL {X  -154.128, Y  +345.852, Z    +0.000, E1   +37.701, E3 +118590.701}
SPL {X  -152.890, Y  +341.633, Z    +0.000, E1   +37.487, E3 +118603.133}
SPL {X  -150.284, Y  +333.893, Z    +0.000, E1   +33.433, E3 +118657.943}
ENDSPLINE

SPLINE
SPL {X  -157.404, Y  +360.095, Z    +0.000, E1   +17.695, E3 +118713.068}
SPL {X  -159.413, Y  +375.108, Z    +0.000, E1    +9.284, E3 +118722.157}
SPL {X  -159.978, Y  +386.135, Z    +0.000, E1    +2.544, E3 +118725.718}
SPL {X  -160.000, Y  +393.708, Z    +0.000, E1    -3.216, E3 +118727.472}
SPL {X  -160.000, Y  +400.474, Z    +0.000, E1    -9.529, E3 +118729.518}
SPL {X  -160.000, Y  +409.652, Z    +0.000, E1   -18.026, E3 +118733.655}
SPL {X  -160.000, Y  +437.804, Z    +0.000, E1   -34.779, E3 +118758.447}
SPL {X  -160.000, Y  +463.067, Z    +0.000, E1   -38.672, E3 +118804.147}
SPL {X  -160.000, Y  +469.167, Z    +0.000, E1   -38.717, E3 +118820.254}
SPL {X  -160.000, Y  +476.691, Z    +0.000, E1   -38.728, E3 +118840.185}
SPL {X  -160.000, Y  +483.419, Z    +0.000, E1   -38.692, E3 +118858.085}
SPL {X  -160.000, Y  +489.013, Z    +0.000, E1   -38.683, E3 +118872.924}
SPL {X  -160.000, Y  +494.786, Z    +0.000, E1   -38.693, E3 +118888.234}
SPL {X  -160.000, Y  +500.108, Z    +0.000, E1   -38.668, E3 +118902.386}
SPL {X  -160.000, Y  +504.903, Z    +0.000, E1   -38.673, E3 +118915.107}
SPL {X  -160.000, Y  +510.180, Z    +0.000, E1   -38.675, E3 +118929.111}
SPL {X  -160.000, Y  +515.083, Z    +0.000, E1   -38.662, E3 +118942.131}
SPL {X  -160.000, Y  +520.479, Z    +0.000, E1   -38.692, E3 +118956.405}
SPL {X  -160.000, Y  +525.998, Z    +0.000, E1   -38.666, E3 +118971.083}
SPL {X  -160.000, Y  +531.341, Z    +0.000, E1   -38.684, E3 +118985.228}
SPL {X  -160.000, Y  +537.313, Z    +0.000, E1   -38.686, E3 +119001.067}
SPL {X  -160.000, Y  +543.203, Z    +0.000, E1   -38.679, E3 +119016.693}
SPL {X  -160.000, Y  +551.201, Z    +0.000, E1   -38.768, E3 +119037.754}
SPL {X  -160.000, Y  +561.335, Z    +0.000, E1   -38.777, E3 +119064.624}
SPL {X  -160.000, Y  +568.812, Z    +0.000, E1   -38.671, E3 +119084.628}
SPL {X  -160.000, Y  +574.116, Z    +0.000, E1   -38.680, E3 +119098.698}
SPL {X  -160.000, Y  +582.193, Z    +0.000, E1   -38.759, E3 +119120.002}
SPL {X  -160.000, Y  +591.932, Z    +0.000, E1   -38.763, E3 +119145.827}
SPL {X  -160.000, Y  +601.488, Z    +0.000, E1   -38.747, E3 +119171.202}
SPL {X  -160.000, Y  +609.161, Z    +0.000, E1   -38.685, E3 +119191.654}
SPL {X  -160.000, Y  +614.445, Z    +0.000, E1   -38.661, E3 +119205.703}
SPL {X  -160.000, Y  +621.895, Z    +0.000, E1   -38.769, E3 +119225.291}
SPL {X  -160.000, Y  +631.692, Z    +0.000, E1   -38.748, E3 +119251.344}
SPL {X  -160.000, Y  +639.246, Z    +0.000, E1   -38.671, E3 +119271.520}
SPL {X  -160.000, Y  +644.827, Z    +0.000, E1   -38.662, E3 +119286.355}
SPL {X  -160.000, Y  +650.491, Z    +0.000, E1   -38.673, E3 +119301.342}
SPL {X  -160.000, Y  +656.011, Z    +0.000, E1   -38.669, E3 +119315.995}
SPL {X  -160.000, Y  +661.156, Z    +0.000, E1   -38.659, E3 +119329.670}
SPL {X  -160.000, Y  +666.701, Z    +0.000, E1   -38.683, E3 +119344.330}
SPL {X  -159.961, Y  +675.011, Z    +0.000, E1   -38.755, E3 +119366.317}
SPL {X  -159.451, Y  +684.743, Z    +0.000, E1   -38.666, E3 +119392.670}
SPL {X  -158.386, Y  +694.170, Z    +0.000, E1   -38.484, E3 +119418.789}
SPL {X  -157.286, Y  +700.846, Z    +0.000, E1   -38.194, E3 +119437.757}
SPL {X  -156.328, Y  +705.580, Z    +0.000, E1   -38.037, E3 +119451.293}
SPL {X  -155.162, Y  +710.549, Z    +0.000, E1   -37.822, E3 +119465.696}
SPL {X  -153.914, Y  +715.210, Z    +0.000, E1   -37.596, E3 +119479.346}
SPL {X  -152.686, Y  +719.322, Z    +0.000, E1   -37.361, E3 +119491.518}
SPL {X  -150.251, Y  +726.496, Z    +0.000, E1   -33.848, E3 +119540.014}
ENDSPLINE

SPLINE
SPL {X  -156.089, Y  +706.662, Z    +0.000, E1   -21.279, E3 +119592.667}
SPL {X  -159.059, Y  +688.824, Z    +0.000, E1   -11.551, E3 +119606.628}
SPL {X  -159.959, Y  +675.119, Z    +0.000, E1    -3.373, E3 +119611.456}
SPL {X  -160.000, Y  +666.447, Z    +0.000, E1    +3.005, E3 +119613.491}
SPL {X  -160.000, Y  +658.774, Z    +0.000, E1   +10.317, E3 +119615.749}
SPL {X  -160.000, Y  +647.765, Z    +0.000, E1   +20.359, E3 +119621.114}
SPL {X  -160.000, Y  +622.607, Z    +0.000, E1   +34.692, E3 +119643.982}
SPL {X  -160.000, Y  +593.120, Z    +0.000, E1   +39.775, E3 +119693.512}
SPL {X  -160.000, Y  +586.287, Z    +0.000, E1   +39.762, E3 +119710.978}
SPL {X  -160.000, Y  +577.753, Z    +0.000, E1   +39.844, E3 +119732.620}
SPL {X  -160.000, Y  +567.367, Z    +0.000, E1   +39.853, E3 +119759.114}
SPL {X  -160.000, Y  +559.466, Z    +0.000, E1   +39.761, E3 +119779.396}
SPL {X  -160.000, Y  +552.914, Z    +0.000, E1   +39.787, E3 +119796.063}
SPL {X  -160.000, Y  +546.390, Z    +0.000, E1   +39.760, E3 +119812.777}
SPL {X  -160.000, Y  +540.123, Z    +0.000, E1   +39.770, E3 +119828.756}
SPL {X  -160.000, Y  +533.658, Z    +0.000, E1   +39.771, E3 +119845.255}
SPL {X  -160.000, Y  +527.046, Z    +0.000, E1   +39.771, E3 +119862.131}
SPL {X  -160.000, Y  +521.063, Z    +0.000, E1   +39.756, E3 +119877.415}
SPL {X  -160.000, Y  +515.110, Z    +0.000, E1   +39.770, E3 +119892.588}
SPL {X  -160.000, Y  +508.717, Z    +0.000, E1   +39.766, E3 +119908.906}
SPL {X  -160.000, Y  +502.133, Z    +0.000, E1   +39.780, E3 +119925.672}
ENDSPLINE

SPLINE
SPL {X  -160.000, Y  +512.949, Z    +0.000, E1   +32.050, E3 +119941.930}
ENDSPLINE

SPLINE
SPL {X  -160.000, Y  +507.092, Z    +0.000, E1   +32.805, E3 +119956.558}
SPL {X  -160.000, Y  +499.824, Z    +0.000, E1   +34.003, E3 +119972.300}
SPL {X  -160.000, Y  +491.367, Z    +0.000, E1   +35.449, E3 +119989.040}
SPL {X  -160.000, Y  +483.082, Z    +0.000, E1   +36.782, E3 +120004.879}
SPL {X  -160.000, Y  +474.521, Z    +0.000, E1   +38.037, E3 +120020.967}
SPL {X  -160.000, Y  +465.343, Z    +0.000, E1   +38.802, E3 +120041.126}
SPL {X  -160.000, Y  +457.266, Z    +0.000, E1   +38.756, E3 +120062.580}
SPL {X  -160.000, Y  +448.553, Z    +0.000, E1   +38.823, E3 +120085.531}
SPL {X  -160.000, Y  +439.425, Z    +0.000, E1   +38.797, E3 +120109.702}
SPL {X  -160.000, Y  +430.351, Z    +0.000, E1   +38.810, E3 +120133.716}
SPL {X  -160.000, Y  +421.477, Z    +0.000, E1   +38.792, E3 +120157.220}
SPL {X  -160.000, Y  +412.292, Z    +0.000, E1   +38.825, E3 +120181.447}
SPL {X  -160.000, Y  +403.281, Z    +0.000, E1   +38.797, E3 +120205.327}
SPL {X  -160.000, Y  +394.948, Z    +0.000, E1   +38.796, E3 +120227.369}
SPL {X  -159.971, Y  +385.741, Z    +0.000, E1   +38.831, E3 +120251.690}
SPL {X  -159.525, Y  +376.478, Z    +0.000, E1   +38.739, E3 +120276.681}
SPL {X  -158.721, Y  +368.613, Z    +0.000, E1   +38.561, E3 +120298.405}
SPL {X  -157.505, Y  +360.654, Z    +0.000, E1   +38.390, E3 +120320.678}
SPL {X  -156.229, Y  +354.269, Z    +0.000, E1   +38.076, E3 +120339.027}
SPL {X  -155.202, Y  +349.910, Z    +0.000, E1   +37.893, E3 +120351.602}
SPL {X  -154.128, Y  +345.852, Z    +0.000, E1   +37.701, E3 +120363.426}
SPL {X  -152.890, Y  +341.633, Z    +0.000, E1   +37.487, E3 +120375.858}
SPL {X  -150.284, Y  +333.893, Z    +0.000, E1   +33.433, E3 +120430.668}
ENDSPLINE

SPLINE
SPL {X  -157.404, Y  +360.095, Z    +0.000, E1   +17.695, E3 +120485.793}
SPL {X  -159.413, Y  +375.108, Z    +0.000, E1    +9.284, E3 +120494.882}
SPL {X  -159.978, Y  +386.135, Z    +0.000, E1    +2.544, E3 +120498.443}
SPL {X  -160.000, Y  +393.708, Z    +0.000, E1    -3.216, E3 +120500.197}
SPL {X  -160.000, Y  +400.474, Z    +0.000, E1    -9.529, E3 +120502.243}
SPL {X  -160.000, Y  +409.652, Z    +0.000, E1   -18.026, E3 +120506.380}
SPL {X  -160.000, Y  +437.804, Z    +0.000, E1   -34.779, E3 +120531.173}
SPL {X  -160.000, Y  +463.067, Z    +0.000, E1   -38.672, E3 +120576.873}
SPL {X  -160.000, Y  +469.167, Z    +0.000, E1   -38.717, E3 +120592.979}
SPL {X  -160.000, Y  +476.691, Z    +0.000, E1   -38.728, E3 +120612.910}
SPL {X  -160.000, Y  +483.419, Z    +0.000, E1   -38.692, E3 +120630.811}
SPL {X  -160.000, Y  +489.013, Z    +0.000, E1   -38.683, E3 +120645.649}
SPL {X  -160.000, Y  +494.786, Z    +0.000, E1   -38.693, E3 +120660.959}
SPL {X  -160.000, Y  +500.108, Z    +0.000, E1   -38.668, E3 +120675.111}
SPL {X  -160.000, Y  +504.903, Z    +0.000, E1   -38.673, E3 +120687.832}
SPL {X  -160.000, Y  +510.180, Z    +0.000, E1   -38.675, E3 +120701.836}
SPL {X  -160.000, Y  +515.083, Z    +0.000, E1   -38.662, E3 +120714.856}
SPL {X  -160.000, Y  +520.479, Z    +0.000, E1   -38.692, E3 +120729.130}
SPL {X  -160.000, Y  +525.998, Z    +0.000, E1   -38.666, E3 +120743.809}
SPL {X  -160.000, Y  +531.341, Z    +0.000, E1   -38.684, E3 +120757.953}
SPL {X  -160.000, Y  +537.313, Z    +0.000, E1   -38.686, E3 +120773.793}
SPL {X  -160.000, Y  +543.203, Z    +0.000, E1   -38.679, E3 +120789.418}
SPL {X  -160.000, Y  +551.201, Z    +0.000, E1   -38.768, E3 +120810.479}
SPL {X  -160.000, Y  +561.335, Z    +0.000, E1   -38.777, E3 +120837.350}
SPL {X  -160.000, Y  +568.812, Z    +0.000, E1   -38.671, E3 +120857.353}
SPL {X  -160.000, Y  +574.116, Z    +0.000, E1   -38.680, E3 +120871.423}
SPL {X  -160.000, Y  +582.193, Z    +0.000, E1   -38.759, E3 +120892.727}
SPL {X  -160.000, Y  +591.932, Z    +0.000, E1   -38.763, E3 +120918.552}
SPL {X  -160.000, Y  +601.488, Z    +0.000, E1   -38.747, E3 +120943.927}
SPL {X  -160.000, Y  +609.161, Z    +0.000, E1   -38.685, E3 +120964.379}
SPL {X  -160.000, Y  +614.445, Z    +0.000, E1   -38.661, E3 +120978.428}
SPL {X  -160.000, Y  +621.895, Z    +0.000, E1   -38.769, E3 +120998.016}
SPL {X  -160.000, Y  +631.692, Z    +0.000, E1   -38.748, E3 +121024.070}
SPL {X  -160.000, Y  +639.246, Z    +0.000, E1   -38.671, E3 +121044.245}
SPL {X  -160.000, Y  +644.827, Z    +0.000, E1   -38.662, E3 +121059.080}
SPL {X  -160.000, Y  +650.491, Z    +0.000, E1   -38.673, E3 +121074.067}
SPL {X  -160.000, Y  +656.011, Z    +0.000, E1   -38.669, E3 +121088.720}
SPL {X  -160.000, Y  +661.156, Z    +0.000, E1   -38.659, E3 +121102.395}
SPL {X  -160.000, Y  +666.701, Z    +0.000, E1   -38.683, E3 +121117.056}
SPL {X  -159.961, Y  +675.011, Z    +0.000, E1   -38.755, E3 +121139.042}
SPL {X  -159.451, Y  +684.743, Z    +0.000, E1   -38.666, E3 +121165.396}
SPL {X  -158.386, Y  +694.170, Z    +0.000, E1   -38.484, E3 +121191.514}
SPL {X  -157.286, Y  +700.846, Z    +0.000, E1   -38.194, E3 +121210.482}
SPL {X  -156.328, Y  +705.580, Z    +0.000, E1   -38.037, E3 +121224.018}
SPL {X  -155.162, Y  +710.549, Z    +0.000, E1   -37.822, E3 +121238.422}
SPL {X  -153.914, Y  +715.210, Z    +0.000, E1   -37.596, E3 +121252.071}
SPL {X  -152.686, Y  +719.322, Z    +0.000, E1   -37.361, E3 +121264.243}
SPL {X  -150.251, Y  +726.496, Z    +0.000, E1   -33.848, E3 +121312.739}
ENDSPLINE

SPLINE
SPL {X  -156.089, Y  +706.662, Z    +0.000, E1   -21.279, E3 +121365.392}
SPL {X  -159.059, Y  +688.824, Z    +0.000, E1   -11.551, E3 +121379.353}
SPL {X  -159.959, Y  +675.119, Z    +0.000, E1    -3.373, E3 +121384.181}
SPL {X  -160.000, Y  +666.447, Z    +0.000, E1    +3.005, E3 +121386.216}
SPL {X  -160.000, Y  +658.774, Z    +0.000, E1   +10.317, E3 +121388.474}
SPL {X  -160.000, Y  +647.765, Z    +0.000, E1   +20.359, E3 +121393.840}
SPL {X  -160.000, Y  +622.607, Z    +0.000, E1   +34.692, E3 +121416.707}
SPL {X  -160.000, Y  +596.106, Z    +0.000, E1   +39.718, E3 +121458.707}
SPL {X  -160.000, Y  +592.273, Z    +0.000, E1   +39.746, E3 +121468.444}
SPL {X  -160.000, Y  +586.287, Z    +0.000, E1   +39.762, E3 +121483.704}
SPL {X  -160.000, Y  +577.753, Z    +0.000, E1   +39.844, E3 +121505.345}
SPL {X  -160.000, Y  +567.367, Z    +0.000, E1   +39.853, E3 +121531.840}
SPL {X  -160.000, Y  +559.466, Z    +0.000, E1   +39.761, E3 +121552.121}
SPL {X  -160.000, Y  +552.914, Z    +0.000, E1   +39.787, E3 +121568.788}
SPL {X  -160.000, Y  +546.390, Z    +0.000, E1   +39.760, E3 +121585.502}
SPL {X  -160.000, Y  +540.123, Z    +0.000, E1   +39.770, E3 +121601.481}
SPL {X  -160.000, Y  +533.658, Z    +0.000, E1   +39.771, E3 +121617.980}
SPL {X  -160.000, Y  +527.046, Z    +0.000, E1   +39.771, E3 +121634.856}
SPL {X  -160.000, Y  +521.063, Z    +0.000, E1   +39.756, E3 +121650.140}
SPL {X  -160.000, Y  +515.110, Z    +0.000, E1   +39.770, E3 +121665.313}
SPL {X  -160.000, Y  +508.717, Z    +0.000, E1   +39.766, E3 +121681.631}
SPL {X  -160.000, Y  +502.133, Z    +0.000, E1   +39.780, E3 +121698.398}
ENDSPLINE

SPLINE
SPL {X  -160.000, Y  +512.949, Z    +0.000, E1   +32.050, E3 +121714.655}
ENDSPLINE

SPLINE
SPL {X  -160.000, Y  +507.092, Z    +0.000, E1   +32.805, E3 +121729.283}
SPL {X  -160.000, Y  +499.824, Z    +0.000, E1   +34.003, E3 +121745.025}
SPL {X  -160.000, Y  +491.367, Z    +0.000, E1   +35.449, E3 +121761.766}
SPL {X  -160.000, Y  +483.082, Z    +0.000, E1   +36.782, E3 +121777.604}
SPL {X  -160.000, Y  +474.521, Z    +0.000, E1   +38.037, E3 +121793.692}
SPL {X  -160.000, Y  +465.343, Z    +0.000, E1   +38.802, E3 +121813.851}
SPL {X  -160.000, Y  +457.266, Z    +0.000, E1   +38.756, E3 +121835.305}
SPL {X  -160.000, Y  +448.553, Z    +0.000, E1   +38.823, E3 +121858.256}
SPL {X  -160.000, Y  +439.425, Z    +0.000, E1   +38.797, E3 +121882.427}
SPL {X  -160.000, Y  +430.351, Z    +0.000, E1   +38.810, E3 +121906.442}
SPL {X  -160.000, Y  +421.477, Z    +0.000, E1   +38.792, E3 +121929.945}
SPL {X  -160.000, Y  +412.292, Z    +0.000, E1   +38.825, E3 +121954.173}
SPL {X  -160.000, Y  +403.281, Z    +0.000, E1   +38.797, E3 +121978.053}
SPL {X  -160.000, Y  +394.948, Z    +0.000, E1   +38.796, E3 +122000.094}
SPL {X  -159.971, Y  +385.741, Z    +0.000, E1   +38.831, E3 +122024.416}
SPL {X  -159.525, Y  +376.478, Z    +0.000, E1   +38.739, E3 +122049.407}
SPL {X  -158.721, Y  +368.613, Z    +0.000, E1   +38.561, E3 +122071.130}
SPL {X  -157.505, Y  +360.654, Z    +0.000, E1   +38.390, E3 +122093.403}
SPL {X  -156.229, Y  +354.269, Z    +0.000, E1   +38.076, E3 +122111.753}
SPL {X  -155.202, Y  +349.910, Z    +0.000, E1   +37.893, E3 +122124.327}
SPL {X  -154.128, Y  +345.852, Z    +0.000, E1   +37.701, E3 +122136.151}
SPL {X  -152.890, Y  +341.633, Z    +0.000, E1   +37.487, E3 +122148.583}
SPL {X  -150.284, Y  +333.893, Z    +0.000, E1   +33.433, E3 +122203.394}
ENDSPLINE

SPLINE
SPL {X  -157.404, Y  +360.095, Z    +0.000, E1   +17.695, E3 +122258.518}
SPL {X  -159.413, Y  +375.108, Z    +0.000, E1    +9.284, E3 +122267.607}
SPL {X  -159.978, Y  +386.135, Z    +0.000, E1    +2.544, E3 +122271.168}
SPL {X  -160.000, Y  +393.708, Z    +0.000, E1    -3.216, E3 +122272.922}
SPL {X  -160.000, Y  +400.474, Z    +0.000, E1    -9.529, E3 +122274.969}
SPL {X  -160.000, Y  +409.652, Z    +0.000, E1   -18.026, E3 +122279.105}
SPL {X  -160.000, Y  +437.804, Z    +0.000, E1   -34.779, E3 +122303.898}
SPL {X  -160.000, Y  +463.067, Z    +0.000, E1   -38.672, E3 +122349.598}
SPL {X  -160.000, Y  +469.167, Z    +0.000, E1   -38.717, E3 +122365.704}
SPL {X  -160.000, Y  +476.691, Z    +0.000, E1   -38.728, E3 +122385.636}
SPL {X  -160.000, Y  +483.419, Z    +0.000, E1   -38.692, E3 +122403.536}
SPL {X  -160.000, Y  +489.013, Z    +0.000, E1   -38.683, E3 +122418.375}
SPL {X  -160.000, Y  +494.786, Z    +0.000, E1   -38.693, E3 +122433.685}
SPL {X  -160.000, Y  +500.108, Z    +0.000, E1   -38.668, E3 +122447.836}
SPL {X  -160.000, Y  +504.903, Z    +0.000, E1   -38.673, E3 +122460.557}
SPL {X  -160.000, Y  +510.180, Z    +0.000, E1   -38.675, E3 +122474.562}
SPL {X  -160.000, Y  +515.083, Z    +0.000, E1   -38.662, E3 +122487.581}
SPL {X  -160.000, Y  +520.479, Z    +0.000, E1   -38.692, E3 +122501.856}
SPL {X  -160.000, Y  +525.998, Z    +0.000, E1   -38.666, E3 +122516.534}
SPL {X  -160.000, Y  +531.341, Z    +0.000, E1   -38.684, E3 +122530.678}
SPL {X  -160.000, Y  +537.313, Z    +0.000, E1   -38.686, E3 +122546.518}
SPL {X  -160.000, Y  +543.203, Z    +0.000, E1   -38.679, E3 +122562.143}
SPL {X  -160.000, Y  +551.201, Z    +0.000, E1   -38.768, E3 +122583.205}
SPL {X  -160.000, Y  +561.335, Z    +0.000, E1   -38.777, E3 +122610.075}
SPL {X  -160.000, Y  +568.812, Z    +0.000, E1   -38.671, E3 +122630.078}
SPL {X  -160.000, Y  +574.116, Z    +0.000, E1   -38.680, E3 +122644.149}
SPL {X  -160.000, Y  +582.193, Z    +0.000, E1   -38.759, E3 +122665.452}
SPL {X  -160.000, Y  +591.932, Z    +0.000, E1   -38.763, E3 +122691.277}
SPL {X  -160.000, Y  +601.488, Z    +0.000, E1   -38.747, E3 +122716.652}
SPL {X  -160.000, Y  +609.161, Z    +0.000, E1   -38.685, E3 +122737.104}
SPL {X  -160.000, Y  +614.445, Z    +0.000, E1   -38.661, E3 +122751.153}
SPL {X  -160.000, Y  +621.895, Z    +0.000, E1   -38.769, E3 +122770.741}
SPL {X  -160.000, Y  +631.692, Z    +0.000, E1   -38.748, E3 +122796.795}
SPL {X  -160.000, Y  +639.246, Z    +0.000, E1   -38.671, E3 +122816.970}
SPL {X  -160.000, Y  +644.827, Z    +0.000, E1   -38.662, E3 +122831.805}
SPL {X  -160.000, Y  +650.491, Z    +0.000, E1   -38.673, E3 +122846.793}
SPL {X  -160.000, Y  +656.011, Z    +0.000, E1   -38.669, E3 +122861.446}
SPL {X  -160.000, Y  +661.156, Z    +0.000, E1   -38.659, E3 +122875.121}
SPL {X  -160.000, Y  +666.701, Z    +0.000, E1   -38.683, E3 +122889.781}
SPL {X  -159.961, Y  +675.011, Z    +0.000, E1   -38.755, E3 +122911.767}
SPL {X  -159.451, Y  +684.743, Z    +0.000, E1   -38.666, E3 +122938.121}
SPL {X  -158.386, Y  +694.170, Z    +0.000, E1   -38.484, E3 +122964.239}
SPL {X  -157.286, Y  +700.846, Z    +0.000, E1   -38.194, E3 +122983.207}
SPL {X  -156.328, Y  +705.580, Z    +0.000, E1   -38.037, E3 +122996.743}
SPL {X  -155.162, Y  +710.549, Z    +0.000, E1   -37.822, E3 +123011.147}
SPL {X  -153.914, Y  +715.210, Z    +0.000, E1   -37.596, E3 +123024.796}
SPL {X  -152.686, Y  +719.322, Z    +0.000, E1   -37.361, E3 +123036.969}
SPL {X  -150.251, Y  +726.496, Z    +0.000, E1   -33.848, E3 +123085.464}
ENDSPLINE

SPLINE
SPL {X  -156.089, Y  +706.662, Z    +0.000, E1   -21.279, E3 +123138.118}
SPL {X  -159.059, Y  +688.824, Z    +0.000, E1   -11.551, E3 +123152.078}
SPL {X  -159.959, Y  +675.119, Z    +0.000, E1    -3.373, E3 +123156.906}
SPL {X  -160.000, Y  +666.447, Z    +0.000, E1    +3.005, E3 +123158.941}
SPL {X  -160.000, Y  +658.774, Z    +0.000, E1   +10.317, E3 +123161.200}
SPL {X  -160.000, Y  +647.765, Z    +0.000, E1   +20.359, E3 +123166.565}
SPL {X  -160.000, Y  +622.607, Z    +0.000, E1   +34.692, E3 +123189.432}
SPL {X  -160.000, Y  +593.120, Z    +0.000, E1   +39.775, E3 +123238.962}
SPL {X  -160.000, Y  +586.287, Z    +0.000, E1   +39.762, E3 +123256.429}
SPL {X  -160.000, Y  +577.753, Z    +0.000, E1   +39.844, E3 +123278.071}
SPL {X  -160.000, Y  +567.367, Z    +0.000, E1   +39.853, E3 +123304.565}
SPL {X  -160.000, Y  +559.466, Z    +0.000, E1   +39.761, E3 +123324.846}
SPL {X  -160.000, Y  +552.914, Z    +0.000, E1   +39.787, E3 +123341.514}
SPL {X  -160.000, Y  +546.390, Z    +0.000, E1   +39.760, E3 +123358.227}
SPL {X  -160.000, Y  +540.123, Z    +0.000, E1   +39.770, E3 +123374.207}
SPL {X  -160.000, Y  +533.658, Z    +0.000, E1   +39.771, E3 +123390.705}
SPL {X  -160.000, Y  +527.046, Z    +0.000, E1   +39.771, E3 +123407.581}
SPL {X  -160.000, Y  +521.063, Z    +0.000, E1   +39.756, E3 +123422.866}
SPL {X  -160.000, Y  +515.110, Z    +0.000, E1   +39.770, E3 +123438.038}
SPL {X  -160.000, Y  +508.717, Z    +0.000, E1   +39.766, E3 +123454.356}
SPL {X  -160.000, Y  +502.133, Z    +0.000, E1   +39.780, E3 +123471.123}
ENDSPLINE

SPLINE
SPL {X  -160.000, Y  +512.949, Z    +0.000, E1   +32.050, E3 +123487.380}
ENDSPLINE

SPLINE
SPL {X  -160.000, Y  +507.092, Z    +0.000, E1   +32.805, E3 +123502.008}
SPL {X  -160.000, Y  +499.824, Z    +0.000, E1   +34.003, E3 +123517.750}
SPL {X  -160.000, Y  +491.367, Z    +0.000, E1   +35.449, E3 +123534.491}
SPL {X  -160.000, Y  +483.082, Z    +0.000, E1   +36.782, E3 +123550.330}
SPL {X  -160.000, Y  +474.521, Z    +0.000, E1   +38.037, E3 +123566.418}
SPL {X  -160.000, Y  +465.343, Z    +0.000, E1   +38.802, E3 +123586.576}
SPL {X  -160.000, Y  +457.266, Z    +0.000, E1   +38.756, E3 +123608.030}
SPL {X  -160.000, Y  +448.553, Z    +0.000, E1   +38.823, E3 +123630.981}
SPL {X  -160.000, Y  +439.425, Z    +0.000, E1   +38.797, E3 +123655.152}
SPL {X  -160.000, Y  +430.351, Z    +0.000, E1   +38.810, E3 +123679.167}
SPL {X  -160.000, Y  +421.477, Z    +0.000, E1   +38.792, E3 +123702.671}
SPL {X  -160.000, Y  +412.292, Z    +0.000, E1   +38.825, E3 +123726.898}
SPL {X  -160.000, Y  +403.281, Z    +0.000, E1   +38.797, E3 +123750.778}
SPL {X  -160.000, Y  +394.948, Z    +0.000, E1   +38.796, E3 +123772.820}
SPL {X  -159.971, Y  +385.741, Z    +0.000, E1   +38.831, E3 +123797.141}
SPL {X  -159.525, Y  +376.478, Z    +0.000, E1   +38.739, E3 +123822.132}
SPL {X  -158.721, Y  +368.613, Z    +0.000, E1   +38.561, E3 +123843.855}
SPL {X  -157.505, Y  +360.654, Z    +0.000, E1   +38.390, E3 +123866.128}
SPL {X  -156.229, Y  +354.269, Z    +0.000, E1   +38.076, E3 +123884.478}
SPL {X  -155.202, Y  +349.910, Z    +0.000, E1   +37.893, E3 +123897.052}
SPL {X  -154.128, Y  +345.852, Z    +0.000, E1   +37.701, E3 +123908.876}
SPL {X  -152.890, Y  +341.633, Z    +0.000, E1   +37.487, E3 +123921.308}
SPL {X  -150.284, Y  +333.893, Z    +0.000, E1   +33.433, E3 +123976.119}
ENDSPLINE

SPLINE
SPL {X  -157.404, Y  +360.095, Z    +0.000, E1   +17.695, E3 +124031.244}
SPL {X  -159.413, Y  +375.108, Z    +0.000, E1    +9.284, E3 +124040.332}
SPL {X  -159.978, Y  +386.135, Z    +0.000, E1    +2.544, E3 +124043.894}
SPL {X  -160.000, Y  +393.708, Z    +0.000, E1    -3.216, E3 +124045.647}
SPL {X  -160.000, Y  +400.474, Z    +0.000, E1    -9.529, E3 +124047.694}
SPL {X  -160.000, Y  +409.652, Z    +0.000, E1   -18.026, E3 +124051.830}
SPL {X  -160.000, Y  +437.804, Z    +0.000, E1   -34.779, E3 +124076.623}
SPL {X  -160.000, Y  +463.067, Z    +0.000, E1   -38.672, E3 +124122.323}
SPL {X  -160.000, Y  +469.167, Z    +0.000, E1   -38.717, E3 +124138.429}
SPL {X  -160.000, Y  +476.691, Z    +0.000, E1   -38.728, E3 +124158.361}
SPL {X  -160.000, Y  +483.419, Z    +0.000, E1   -38.692, E3 +124176.261}
SPL {X  -160.000, Y  +489.013, Z    +0.000, E1   -38.683, E3 +124191.100}
SPL {X  -160.000, Y  +494.786, Z    +0.000, E1   -38.693, E3 +124206.410}
SPL {X  -160.000, Y  +500.108, Z    +0.000, E1   -38.668, E3 +124220.561}
SPL {X  -160.000, Y  +504.903, Z    +0.000, E1   -38.673, E3 +124233.282}
SPL {X  -160.000, Y  +510.180, Z    +0.000, E1   -38.675, E3 +124247.287}
SPL {X  -160.000, Y  +515.083, Z    +0.000, E1   -38.662, E3 +124260.306}
SPL {X  -160.000, Y  +520.479, Z    +0.000, E1   -38.692, E3 +124274.581}
SPL {X  -160.000, Y  +525.998, Z    +0.000, E1   -38.666, E3 +124289.259}
SPL {X  -160.000, Y  +531.341, Z    +0.000, E1   -38.684, E3 +124303.403}
SPL {X  -160.000, Y  +537.313, Z    +0.000, E1   -38.686, E3 +124319.243}
SPL {X  -160.000, Y  +543.203, Z    +0.000, E1   -38.679, E3 +124334.869}
SPL {X  -160.000, Y  +551.201, Z    +0.000, E1   -38.768, E3 +124355.930}
SPL {X  -160.000, Y  +561.335, Z    +0.000, E1   -38.777, E3 +124382.800}
SPL {X  -160.000, Y  +568.812, Z    +0.000, E1   -38.671, E3 +124402.803}
SPL {X  -160.000, Y  +574.116, Z    +0.000, E1   -38.680, E3 +124416.874}
SPL {X  -160.000, Y  +582.193, Z    +0.000, E1   -38.759, E3 +124438.177}
SPL {X  -160.000, Y  +591.932, Z    +0.000, E1   -38.763, E3 +124464.002}
SPL {X  -160.000, Y  +601.488, Z    +0.000, E1   -38.747, E3 +124489.378}
SPL {X  -160.000, Y  +609.161, Z    +0.000, E1   -38.685, E3 +124509.829}
SPL {X  -160.000, Y  +614.445, Z    +0.000, E1   -38.661, E3 +124523.878}
SPL {X  -160.000, Y  +621.895, Z    +0.000, E1   -38.769, E3 +124543.467}
SPL {X  -160.000, Y  +631.692, Z    +0.000, E1   -38.748, E3 +124569.520}
SPL {X  -160.000, Y  +639.246, Z    +0.000, E1   -38.671, E3 +124589.696}
SPL {X  -160.000, Y  +644.827, Z    +0.000, E1   -38.662, E3 +124604.530}
SPL {X  -160.000, Y  +650.491, Z    +0.000, E1   -38.673, E3 +124619.518}
SPL {X  -160.000, Y  +656.011, Z    +0.000, E1   -38.669, E3 +124634.171}
SPL {X  -160.000, Y  +661.156, Z    +0.000, E1   -38.659, E3 +124647.846}
SPL {X  -160.000, Y  +666.701, Z    +0.000, E1   -38.683, E3 +124662.506}
SPL {X  -159.961, Y  +675.011, Z    +0.000, E1   -38.755, E3 +124684.493}
SPL {X  -159.451, Y  +684.743, Z    +0.000, E1   -38.666, E3 +124710.846}
SPL {X  -158.386, Y  +694.170, Z    +0.000, E1   -38.484, E3 +124736.965}
SPL {X  -157.286, Y  +700.846, Z    +0.000, E1   -38.194, E3 +124755.932}
SPL {X  -156.328, Y  +705.580, Z    +0.000, E1   -38.037, E3 +124769.468}
SPL {X  -155.162, Y  +710.549, Z    +0.000, E1   -37.822, E3 +124783.872}
SPL {X  -153.914, Y  +715.210, Z    +0.000, E1   -37.596, E3 +124797.522}
SPL {X  -152.686, Y  +719.322, Z    +0.000, E1   -37.361, E3 +124809.694}
SPL {X  -150.251, Y  +726.496, Z    +0.000, E1   -33.848, E3 +124858.190}
ENDSPLINE

SPLINE
SPL {X  -156.089, Y  +706.662, Z    +0.000, E1   -21.279, E3 +124910.843}
SPL {X  -159.059, Y  +688.824, Z    +0.000, E1   -11.551, E3 +124924.803}
SPL {X  -159.959, Y  +675.119, Z    +0.000, E1    -3.373, E3 +124929.632}
SPL {X  -160.000, Y  +666.447, Z    +0.000, E1    +3.005, E3 +124931.666}
SPL {X  -160.000, Y  +658.774, Z    +0.000, E1   +10.317, E3 +124933.925}
SPL {X  -160.000, Y  +647.765, Z    +0.000, E1   +20.359, E3 +124939.290}
SPL {X  -160.000, Y  +622.607, Z    +0.000, E1   +34.692, E3 +124962.157}
SPL {X  -160.000, Y  +596.106, Z    +0.000, E1   +39.718, E3 +125004.157}
SPL {X  -160.000, Y  +592.273, Z    +0.000, E1   +39.746, E3 +125013.895}
SPL {X  -160.000, Y  +586.287, Z    +0.000, E1   +39.762, E3 +125029.154}
SPL {X  -160.000, Y  +577.753, Z    +0.000, E1   +39.844, E3 +125050.796}
SPL {X  -160.000, Y  +567.367, Z    +0.000, E1   +39.853, E3 +125077.290}
SPL {X  -160.000, Y  +559.466, Z    +0.000, E1   +39.761, E3 +125097.571}
SPL {X  -160.000, Y  +552.914, Z    +0.000, E1   +39.787, E3 +125114.239}
SPL {X  -160.000, Y  +546.390, Z    +0.000, E1   +39.760, E3 +125130.953}
SPL {X  -160.000, Y  +540.123, Z    +0.000, E1   +39.770, E3 +125146.932}
SPL {X  -160.000, Y  +533.658, Z    +0.000, E1   +39.771, E3 +125163.430}
SPL {X  -160.000, Y  +527.046, Z    +0.000, E1   +39.771, E3 +125180.306}
SPL {X  -160.000, Y  +521.063, Z    +0.000, E1   +39.756, E3 +125195.591}
SPL {X  -160.000, Y  +515.110, Z    +0.000, E1   +39.770, E3 +125210.763}
SPL {X  -160.000, Y  +508.717, Z    +0.000, E1   +39.766, E3 +125227.082}
SPL {X  -160.000, Y  +502.133, Z    +0.000, E1   +39.780, E3 +125243.848}
ENDSPLINE

SPLINE
SPL {X  -160.000, Y  +512.949, Z    +0.000, E1   +32.050, E3 +125260.105}
ENDSPLINE

SPLINE
SPL {X  -160.000, Y  +507.092, Z    +0.000, E1   +32.805, E3 +125274.734}
SPL {X  -160.000, Y  +499.824, Z    +0.000, E1   +34.003, E3 +125290.476}
SPL {X  -160.000, Y  +491.367, Z    +0.000, E1   +35.449, E3 +125307.216}
SPL {X  -160.000, Y  +483.082, Z    +0.000, E1   +36.782, E3 +125323.055}
SPL {X  -160.000, Y  +474.521, Z    +0.000, E1   +38.037, E3 +125339.143}
SPL {X  -160.000, Y  +465.343, Z    +0.000, E1   +38.802, E3 +125359.302}
SPL {X  -160.000, Y  +457.266, Z    +0.000, E1   +38.756, E3 +125380.755}
SPL {X  -160.000, Y  +448.553, Z    +0.000, E1   +38.823, E3 +125403.706}
SPL {X  -160.000, Y  +439.425, Z    +0.000, E1   +38.797, E3 +125427.877}
SPL {X  -160.000, Y  +430.351, Z    +0.000, E1   +38.810, E3 +125451.892}
SPL {X  -160.000, Y  +421.477, Z    +0.000, E1   +38.792, E3 +125475.396}
SPL {X  -160.000, Y  +412.292, Z    +0.000, E1   +38.825, E3 +125499.623}
SPL {X  -160.000, Y  +403.281, Z    +0.000, E1   +38.797, E3 +125523.503}
SPL {X  -160.000, Y  +394.948, Z    +0.000, E1   +38.796, E3 +125545.545}
SPL {X  -159.971, Y  +385.741, Z    +0.000, E1   +38.831, E3 +125569.866}
SPL {X  -159.525, Y  +376.478, Z    +0.000, E1   +38.739, E3 +125594.857}
SPL {X  -158.721, Y  +368.613, Z    +0.000, E1   +38.561, E3 +125616.580}
SPL {X  -157.505, Y  +360.654, Z    +0.000, E1   +38.390, E3 +125638.853}
SPL {X  -156.229, Y  +354.269, Z    +0.000, E1   +38.076, E3 +125657.203}
SPL {X  -155.202, Y  +349.910, Z    +0.000, E1   +37.893, E3 +125669.778}
SPL {X  -154.128, Y  +345.852, Z    +0.000, E1   +37.701, E3 +125681.602}
SPL {X  -152.890, Y  +341.633, Z    +0.000, E1   +37.487, E3 +125694.034}
SPL {X  -150.284, Y  +333.893, Z    +0.000, E1   +33.433, E3 +125748.844}
ENDSPLINE

SPLINE
SPL {X  -157.404, Y  +360.095, Z    +0.000, E1   +17.695, E3 +125803.969}
SPL {X  -159.413, Y  +375.108, Z    +0.000, E1    +9.284, E3 +125813.058}
SPL {X  -159.978, Y  +386.135, Z    +0.000, E1    +2.544, E3 +125816.619}
SPL {X  -160.000, Y  +393.708, Z    +0.000, E1    -3.216, E3 +125818.373}
SPL {X  -160.000, Y  +400.474, Z    +0.000, E1    -9.529, E3 +125820.419}
SPL {X  -160.000, Y  +409.652, Z    +0.000, E1   -18.026, E3 +125824.556}
SPL {X  -160.000, Y  +437.804, Z    +0.000, E1   -34.779, E3 +125849.348}
SPL {X  -160.000, Y  +463.067, Z    +0.000, E1   -38.672, E3 +125895.048}
SPL {X  -160.000, Y  +469.167, Z    +0.000, E1   -38.717, E3 +125911.155}
SPL {X  -160.000, Y  +476.691, Z    +0.000, E1   -38.728, E3 +125931.086}
SPL {X  -160.000, Y  +483.419, Z    +0.000, E1   -38.692, E3 +125948.986}
SPL {X  -160.000, Y  +489.013, Z    +0.000, E1   -38.683, E3 +125963.825}
SPL {X  -160.000, Y  +494.786, Z    +0.000, E1   -38.693, E3 +125979.135}
SPL {X  -160.000, Y  +500.108, Z    +0.000, E1   -38.668, E3 +125993.287}
SPL {X  -160.000, Y  +504.903, Z    +0.000, E1   -38.673, E3 +126006.008}
SPL {X  -160.000, Y  +510.180, Z    +0.000, E1   -38.675, E3 +126020.012}
SPL {X  -160.000, Y  +515.083, Z    +0.000, E1   -38.662, E3 +126033.032}
SPL {X  -160.000, Y  +520.479, Z    +0.000, E1   -38.692, E3 +126047.306}
SPL {X  -160.000, Y  +525.998, Z    +0.000, E1   -38.666, E3 +126061.984}
SPL {X  -160.000, Y  +531.341, Z    +0.000, E1   -38.684, E3 +126076.128}
SPL {X  -160.000, Y  +537.313, Z    +0.000, E1   -38.686, E3 +126091.968}
SPL {X  -160.000, Y  +543.203, Z    +0.000, E1   -38.679, E3 +126107.594}
SPL {X  -160.000, Y  +551.201, Z    +0.000, E1   -38.768, E3 +126128.655}
SPL {X  -160.000, Y  +561.335, Z    +0.000, E1   -38.777, E3 +126155.525}
SPL {X  -160.000, Y  +568.812, Z    +0.000, E1   -38.671, E3 +126175.529}
SPL {X  -160.000, Y  +574.116, Z    +0.000, E1   -38.680, E3 +126189.599}
SPL {X  -160.000, Y  +582.193, Z    +0.000, E1   -38.759, E3 +126210.903}
SPL {X  -160.000, Y  +591.932, Z    +0.000, E1   -38.763, E3 +126236.728}
SPL {X  -160.000, Y  +601.488, Z    +0.000, E1   -38.747, E3 +126262.103}
SPL {X  -160.000, Y  +609.161, Z    +0.000, E1   -38.685, E3 +126282.555}
SPL {X  -160.000, Y  +614.445, Z    +0.000, E1   -38.661, E3 +126296.604}
SPL {X  -160.000, Y  +621.895, Z    +0.000, E1   -38.769, E3 +126316.192}
SPL {X  -160.000, Y  +631.692, Z    +0.000, E1   -38.748, E3 +126342.245}
SPL {X  -160.000, Y  +639.246, Z    +0.000, E1   -38.671, E3 +126362.421}
SPL {X  -160.000, Y  +644.827, Z    +0.000, E1   -38.662, E3 +126377.256}
SPL {X  -160.000, Y  +650.491, Z    +0.000, E1   -38.673, E3 +126392.243}
SPL {X  -160.000, Y  +656.011, Z    +0.000, E1   -38.669, E3 +126406.896}
SPL {X  -160.000, Y  +661.156, Z    +0.000, E1   -38.659, E3 +126420.571}
SPL {X  -160.000, Y  +666.701, Z    +0.000, E1   -38.683, E3 +126435.231}
SPL {X  -159.961, Y  +675.011, Z    +0.000, E1   -38.755, E3 +126457.218}
SPL {X  -159.451, Y  +684.743, Z    +0.000, E1   -38.666, E3 +126483.571}
SPL {X  -158.386, Y  +694.170, Z    +0.000, E1   -38.484, E3 +126509.690}
SPL {X  -157.286, Y  +700.846, Z    +0.000, E1   -38.194, E3 +126528.658}
SPL {X  -156.328, Y  +705.580, Z    +0.000, E1   -38.037, E3 +126542.194}
SPL {X  -155.162, Y  +710.549, Z    +0.000, E1   -37.822, E3 +126556.597}
SPL {X  -153.914, Y  +715.210, Z    +0.000, E1   -37.596, E3 +126570.247}
SPL {X  -152.686, Y  +719.322, Z    +0.000, E1   -37.361, E3 +126582.419}
SPL {X  -150.251, Y  +726.496, Z    +0.000, E1   -33.848, E3 +126630.915}
ENDSPLINE

SPLINE
SPL {X  -156.089, Y  +706.662, Z    +0.000, E1   -21.279, E3 +126683.568}
SPL {X  -159.059, Y  +688.824, Z    +0.000, E1   -11.551, E3 +126697.529}
SPL {X  -159.959, Y  +675.119, Z    +0.000, E1    -3.373, E3 +126702.357}
SPL {X  -160.000, Y  +666.447, Z    +0.000, E1    +3.005, E3 +126704.392}
SPL {X  -160.000, Y  +658.774, Z    +0.000, E1   +10.317, E3 +126706.650}
SPL {X  -160.000, Y  +647.765, Z    +0.000, E1   +20.359, E3 +126712.015}
SPL {X  -160.000, Y  +622.607, Z    +0.000, E1   +34.692, E3 +126734.883}
SPL {X  -160.000, Y  +593.120, Z    +0.000, E1   +39.775, E3 +126784.413}
SPL {X  -160.000, Y  +586.287, Z    +0.000, E1   +39.762, E3 +126801.879}
SPL {X  -160.000, Y  +577.753, Z    +0.000, E1   +39.844, E3 +126823.521}
SPL {X  -160.000, Y  +567.367, Z    +0.000, E1   +39.853, E3 +126850.015}
SPL {X  -160.000, Y  +559.466, Z    +0.000, E1   +39.761, E3 +126870.297}
SPL {X  -160.000, Y  +552.914, Z    +0.000, E1   +39.787, E3 +126886.964}
SPL {X  -160.000, Y  +546.390, Z    +0.000, E1   +39.760, E3 +126903.678}
SPL {X  -160.000, Y  +540.123, Z    +0.000, E1   +39.770, E3 +126919.657}
SPL {X  -160.000, Y  +533.658, Z    +0.000, E1   +39.771, E3 +126936.156}
SPL {X  -160.000, Y  +527.046, Z    +0.000, E1   +39.771, E3 +126953.031}
SPL {X  -160.000, Y  +521.063, Z    +0.000, E1   +39.756, E3 +126968.316}
SPL {X  -160.000, Y  +515.110, Z    +0.000, E1   +39.770, E3 +126983.488}
SPL {X  -160.000, Y  +508.717, Z    +0.000, E1   +39.766, E3 +126999.807}
SPL {X  -160.000, Y  +502.133, Z    +0.000, E1   +39.780, E3 +127016.573}
ENDSPLINE

SPLINE
SPL {X  -160.000, Y  +512.949, Z    +0.000, E1   +32.050, E3 +127032.831}
ENDSPLINE

SPLINE
SPL {X  -160.000, Y  +507.092, Z    +0.000, E1   +32.805, E3 +127047.459}
SPL {X  -160.000, Y  +499.824, Z    +0.000, E1   +34.003, E3 +127063.201}
SPL {X  -160.000, Y  +491.367, Z    +0.000, E1   +35.449, E3 +127079.941}
SPL {X  -160.000, Y  +483.082, Z    +0.000, E1   +36.782, E3 +127095.780}
SPL {X  -160.000, Y  +474.521, Z    +0.000, E1   +38.037, E3 +127111.868}
SPL {X  -160.000, Y  +465.343, Z    +0.000, E1   +38.802, E3 +127132.027}
SPL {X  -160.000, Y  +457.266, Z    +0.000, E1   +38.756, E3 +127153.481}
SPL {X  -160.000, Y  +448.553, Z    +0.000, E1   +38.823, E3 +127176.432}
SPL {X  -160.000, Y  +439.425, Z    +0.000, E1   +38.797, E3 +127200.603}
SPL {X  -160.000, Y  +430.351, Z    +0.000, E1   +38.810, E3 +127224.617}
SPL {X  -160.000, Y  +421.477, Z    +0.000, E1   +38.792, E3 +127248.121}
SPL {X  -160.000, Y  +412.292, Z    +0.000, E1   +38.825, E3 +127272.348}
SPL {X  -160.000, Y  +403.281, Z    +0.000, E1   +38.797, E3 +127296.228}
SPL {X  -160.000, Y  +394.948, Z    +0.000, E1   +38.796, E3 +127318.270}
SPL {X  -159.971, Y  +385.741, Z    +0.000, E1   +38.831, E3 +127342.591}
SPL {X  -159.525, Y  +376.478, Z    +0.000, E1   +38.739, E3 +127367.582}
SPL {X  -158.721, Y  +368.613, Z    +0.000, E1   +38.561, E3 +127389.305}
SPL {X  -157.505, Y  +360.654, Z    +0.000, E1   +38.390, E3 +127411.579}
SPL {X  -156.229, Y  +354.269, Z    +0.000, E1   +38.076, E3 +127429.928}
SPL {X  -155.202, Y  +349.910, Z    +0.000, E1   +37.893, E3 +127442.503}
SPL {X  -154.128, Y  +345.852, Z    +0.000, E1   +37.701, E3 +127454.327}
SPL {X  -152.890, Y  +341.633, Z    +0.000, E1   +37.487, E3 +127466.759}
SPL {X  -150.284, Y  +333.893, Z    +0.000, E1   +33.433, E3 +127521.569}
ENDSPLINE

SPLINE
SPL {X  -157.404, Y  +360.095, Z    +0.000, E1   +17.695, E3 +127576.694}
SPL {X  -159.413, Y  +375.108, Z    +0.000, E1    +9.284, E3 +127585.783}
SPL {X  -159.978, Y  +386.135, Z    +0.000, E1    +2.544, E3 +127589.344}
SPL {X  -160.000, Y  +393.708, Z    +0.000, E1    -3.216, E3 +127591.098}
SPL {X  -160.000, Y  +400.474, Z    +0.000, E1    -9.529, E3 +127593.144}
SPL {X  -160.000, Y  +409.652, Z    +0.000, E1   -18.026, E3 +127597.281}
SPL {X  -160.000, Y  +437.804, Z    +0.000, E1   -34.779, E3 +127622.074}
SPL {X  -160.000, Y  +463.067, Z    +0.000, E1   -38.672, E3 +127667.774}
SPL {X  -160.000, Y  +469.167, Z    +0.000, E1   -38.717, E3 +127683.880}
SPL {X  -160.000, Y  +476.691, Z    +0.000, E1   -38.728, E3 +127703.811}
SPL {X  -160.000, Y  +483.419, Z    +0.000, E1   -38.692, E3 +127721.712}
SPL {X  -160.000, Y  +489.013, Z    +0.000, E1   -38.683, E3 +127736.550}
SPL {X  -160.000, Y  +494.786, Z    +0.000, E1   -38.693, E3 +127751.860}
SPL {X  -160.000, Y  +500.108, Z    +0.000, E1   -38.668, E3 +127766.012}
SPL {X  -160.000, Y  +504.903, Z    +0.000, E1   -38.673, E3 +127778.733}
SPL {X  -160.000, Y  +510.180, Z    +0.000, E1   -38.675, E3 +127792.737}
SPL {X  -160.000, Y  +515.083, Z    +0.000, E1   -38.662, E3 +127805.757}
SPL {X  -160.000, Y  +520.479, Z    +0.000, E1   -38.692, E3 +127820.031}
SPL {X  -160.000, Y  +525.998, Z    +0.000, E1   -38.666, E3 +127834.710}
SPL {X  -160.000, Y  +531.341, Z    +0.000, E1   -38.684, E3 +127848.854}
SPL {X  -160.000, Y  +537.313, Z    +0.000, E1   -38.686, E3 +127864.694}
SPL {X  -160.000, Y  +543.203, Z    +0.000, E1   -38.679, E3 +127880.319}
SPL {X  -160.000, Y  +551.201, Z    +0.000, E1   -38.768, E3 +127901.380}
SPL {X  -160.000, Y  +561.335, Z    +0.000, E1   -38.777, E3 +127928.251}
SPL {X  -160.000, Y  +568.812, Z    +0.000, E1   -38.671, E3 +127948.254}
SPL {X  -160.000, Y  +574.116, Z    +0.000, E1   -38.680, E3 +127962.324}
SPL {X  -160.000, Y  +582.193, Z    +0.000, E1   -38.759, E3 +127983.628}
SPL {X  -160.000, Y  +591.932, Z    +0.000, E1   -38.763, E3 +128009.453}
SPL {X  -160.000, Y  +601.488, Z    +0.000, E1   -38.747, E3 +128034.828}
SPL {X  -160.000, Y  +609.161, Z    +0.000, E1   -38.685, E3 +128055.280}
SPL {X  -160.000, Y  +614.445, Z    +0.000, E1   -38.661, E3 +128069.329}
SPL {X  -160.000, Y  +621.895, Z    +0.000, E1   -38.769, E3 +128088.917}
SPL {X  -160.000, Y  +631.692, Z    +0.000, E1   -38.748, E3 +128114.970}
SPL {X  -160.000, Y  +639.246, Z    +0.000, E1   -38.671, E3 +128135.146}
SPL {X  -160.000, Y  +644.827, Z    +0.000, E1   -38.662, E3 +128149.981}
SPL {X  -160.000, Y  +650.491, Z    +0.000, E1   -38.673, E3 +128164.968}
SPL {X  -160.000, Y  +656.011, Z    +0.000, E1   -38.669, E3 +128179.621}
SPL {X  -160.000, Y  +661.156, Z    +0.000, E1   -38.659, E3 +128193.296}
SPL {X  -160.000, Y  +666.701, Z    +0.000, E1   -38.683, E3 +128207.957}
SPL {X  -159.961, Y  +675.011, Z    +0.000, E1   -38.755, E3 +128229.943}
SPL {X  -159.451, Y  +684.743, Z    +0.000, E1   -38.666, E3 +128256.297}
SPL {X  -158.386, Y  +694.170, Z    +0.000, E1   -38.484, E3 +128282.415}
SPL {X  -157.286, Y  +700.846, Z    +0.000, E1   -38.194, E3 +128301.383}
SPL {X  -156.328, Y  +705.580, Z    +0.000, E1   -38.037, E3 +128314.919}
SPL {X  -155.162, Y  +710.549, Z    +0.000, E1   -37.822, E3 +128329.323}
SPL {X  -153.914, Y  +715.210, Z    +0.000, E1   -37.596, E3 +128342.972}
SPL {X  -152.686, Y  +719.322, Z    +0.000, E1   -37.361, E3 +128355.144}
SPL {X  -150.251, Y  +726.496, Z    +0.000, E1   -33.848, E3 +128403.640}
ENDSPLINE

SPLINE
SPL {X  -156.089, Y  +706.662, Z    +0.000, E1   -21.279, E3 +128456.293}
SPL {X  -159.059, Y  +688.824, Z    +0.000, E1   -11.551, E3 +128470.254}
SPL {X  -159.959, Y  +675.119, Z    +0.000, E1    -3.373, E3 +128475.082}
SPL {X  -160.000, Y  +666.447, Z    +0.000, E1    +3.005, E3 +128477.117}
SPL {X  -160.000, Y  +658.774, Z    +0.000, E1   +10.317, E3 +128479.375}
SPL {X  -160.000, Y  +647.765, Z    +0.000, E1   +20.359, E3 +128484.741}
SPL {X  -160.000, Y  +622.607, Z    +0.000, E1   +34.692, E3 +128507.608}
SPL {X  -160.000, Y  +596.106, Z    +0.000, E1   +39.718, E3 +128549.608}
SPL {X  -160.000, Y  +592.273, Z    +0.000, E1   +39.746, E3 +128559.345}
SPL {X  -160.000, Y  +586.287, Z    +0.000, E1   +39.762, E3 +128574.605}
SPL {X  -160.000, Y  +577.753, Z    +0.000, E1   +39.844, E3 +128596.246}
SPL {X  -160.000, Y  +567.367, Z    +0.000, E1   +39.853, E3 +128622.741}
SPL {X  -160.000, Y  +559.466, Z    +0.000, E1   +39.761, E3 +128643.022}
SPL {X  -160.000, Y  +552.914, Z    +0.000, E1   +39.787, E3 +128659.689}
SPL {X  -160.000, Y  +546.390, Z    +0.000, E1   +39.760, E3 +128676.403}
SPL {X  -160.000, Y  +540.123, Z    +0.000, E1   +39.770, E3 +128692.382}
SPL {X  -160.000, Y  +533.658, Z    +0.000, E1   +39.771, E3 +128708.881}
SPL {X  -160.000, Y  +527.046, Z    +0.000, E1   +39.771, E3 +128725.757}
SPL {X  -160.000, Y  +521.063, Z    +0.000, E1   +39.756, E3 +128741.041}
SPL {X  -160.000, Y  +515.110, Z    +0.000, E1   +39.770, E3 +128756.214}
SPL {X  -160.000, Y  +508.717, Z    +0.000, E1   +39.766, E3 +128772.532}
SPL {X  -160.000, Y  +502.133, Z    +0.000, E1   +39.780, E3 +128789.299}
ENDSPLINE

SPLINE
SPL {X  -160.000, Y  +512.949, Z    +0.000, E1   +32.050, E3 +128805.556}
ENDSPLINE

SPLINE
SPL {X  -160.000, Y  +507.092, Z    +0.000, E1   +32.805, E3 +128820.184}
SPL {X  -160.000, Y  +499.824, Z    +0.000, E1   +34.003, E3 +128835.926}
SPL {X  -160.000, Y  +491.367, Z    +0.000, E1   +35.449, E3 +128852.667}
SPL {X  -160.000, Y  +483.082, Z    +0.000, E1   +36.782, E3 +128868.505}
SPL {X  -160.000, Y  +474.521, Z    +0.000, E1   +38.037, E3 +128884.593}
SPL {X  -160.000, Y  +465.343, Z    +0.000, E1   +38.802, E3 +128904.752}
SPL {X  -160.000, Y  +457.266, Z    +0.000, E1   +38.756, E3 +128926.206}
SPL {X  -160.000, Y  +448.553, Z    +0.000, E1   +38.823, E3 +128949.157}
SPL {X  -160.000, Y  +439.425, Z    +0.000, E1   +38.797, E3 +128973.328}
SPL {X  -160.000, Y  +430.351, Z    +0.000, E1   +38.810, E3 +128997.343}
SPL {X  -160.000, Y  +421.477, Z    +0.000, E1   +38.792, E3 +129020.846}
SPL {X  -160.000, Y  +412.292, Z    +0.000, E1   +38.825, E3 +129045.074}
SPL {X  -160.000, Y  +403.281, Z    +0.000, E1   +38.797, E3 +129068.954}
SPL {X  -160.000, Y  +394.948, Z    +0.000, E1   +38.796, E3 +129090.995}
SPL {X  -159.971, Y  +385.741, Z    +0.000, E1   +38.831, E3 +129115.317}
SPL {X  -159.525, Y  +376.478, Z    +0.000, E1   +38.739, E3 +129140.308}
SPL {X  -158.721, Y  +368.613, Z    +0.000, E1   +38.561, E3 +129162.031}
SPL {X  -157.505, Y  +360.654, Z    +0.000, E1   +38.390, E3 +129184.304}
SPL {X  -156.229, Y  +354.269, Z    +0.000, E1   +38.076, E3 +129202.654}
SPL {X  -155.202, Y  +349.910, Z    +0.000, E1   +37.893, E3 +129215.228}
SPL {X  -154.128, Y  +345.852, Z    +0.000, E1   +37.701, E3 +129227.052}
SPL {X  -152.890, Y  +341.633, Z    +0.000, E1   +37.487, E3 +129239.484}
SPL {X  -150.284, Y  +333.893, Z    +0.000, E1   +33.433, E3 +129294.294}
ENDSPLINE

SPLINE
SPL {X  -157.404, Y  +360.095, Z    +0.000, E1   +17.695, E3 +129349.419}
SPL {X  -159.413, Y  +375.108, Z    +0.000, E1    +9.284, E3 +129358.508}
SPL {X  -159.978, Y  +386.135, Z    +0.000, E1    +2.544, E3 +129362.069}
SPL {X  -160.000, Y  +393.708, Z    +0.000, E1    -3.216, E3 +129363.823}
SPL {X  -160.000, Y  +400.474, Z    +0.000, E1    -9.529, E3 +129365.870}
SPL {X  -160.000, Y  +409.652, Z    +0.000, E1   -18.026, E3 +129370.006}
SPL {X  -160.000, Y  +437.804, Z    +0.000, E1   -34.779, E3 +129394.799}
SPL {X  -160.000, Y  +463.067, Z    +0.000, E1   -38.672, E3 +129440.499}
SPL {X  -160.000, Y  +469.167, Z    +0.000, E1   -38.717, E3 +129456.605}
SPL {X  -160.000, Y  +476.691, Z    +0.000, E1   -38.728, E3 +129476.537}
SPL {X  -160.000, Y  +483.419, Z    +0.000, E1   -38.692, E3 +129494.437}
SPL {X  -160.000, Y  +489.013, Z    +0.000, E1   -38.683, E3 +129509.276}
SPL {X  -160.000, Y  +494.786, Z    +0.000, E1   -38.693, E3 +129524.586}
SPL {X  -160.000, Y  +500.108, Z    +0.000, E1   -38.668, E3 +129538.737}
SPL {X  -160.000, Y  +504.903, Z    +0.000, E1   -38.673, E3 +129551.458}
SPL {X  -160.000, Y  +510.180, Z    +0.000, E1   -38.675, E3 +129565.463}
SPL {X  -160.000, Y  +515.083, Z    +0.000, E1   -38.662, E3 +129578.482}
SPL {X  -160.000, Y  +520.479, Z    +0.000, E1   -38.692, E3 +129592.757}
SPL {X  -160.000, Y  +525.998, Z    +0.000, E1   -38.666, E3 +129607.435}
SPL {X  -160.000, Y  +531.341, Z    +0.000, E1   -38.684, E3 +129621.579}
SPL {X  -160.000, Y  +537.313, Z    +0.000, E1   -38.686, E3 +129637.419}
SPL {X  -160.000, Y  +543.203, Z    +0.000, E1   -38.679, E3 +129653.044}
SPL {X  -160.000, Y  +551.201, Z    +0.000, E1   -38.768, E3 +129674.106}
SPL {X  -160.000, Y  +561.335, Z    +0.000, E1   -38.777, E3 +129700.976}
SPL {X  -160.000, Y  +568.812, Z    +0.000, E1   -38.671, E3 +129720.979}
SPL {X  -160.000, Y  +574.116, Z    +0.000, E1   -38.680, E3 +129735.050}
SPL {X  -160.000, Y  +582.193, Z    +0.000, E1   -38.759, E3 +129756.353}
SPL {X  -160.000, Y  +591.932, Z    +0.000, E1   -38.763, E3 +129782.178}
SPL {X  -160.000, Y  +601.488, Z    +0.000, E1   -38.747, E3 +129807.553}
SPL {X  -160.000, Y  +609.161, Z    +0.000, E1   -38.685, E3 +129828.005}
SPL {X  -160.000, Y  +614.445, Z    +0.000, E1   -38.661, E3 +129842.054}
SPL {X  -160.000, Y  +621.895, Z    +0.000, E1   -38.769, E3 +129861.642}
SPL {X  -160.000, Y  +631.692, Z    +0.000, E1   -38.748, E3 +129887.696}
SPL {X  -160.000, Y  +639.246, Z    +0.000, E1   -38.671, E3 +129907.871}
SPL {X  -160.000, Y  +644.827, Z    +0.000, E1   -38.662, E3 +129922.706}
SPL {X  -160.000, Y  +650.491, Z    +0.000, E1   -38.673, E3 +129937.694}
SPL {X  -160.000, Y  +656.011, Z    +0.000, E1   -38.669, E3 +129952.347}
SPL {X  -160.000, Y  +661.156, Z    +0.000, E1   -38.659, E3 +129966.022}
SPL {X  -160.000, Y  +666.701, Z    +0.000, E1   -38.683, E3 +129980.682}
SPL {X  -159.961, Y  +675.011, Z    +0.000, E1   -38.755, E3 +130002.668}
SPL {X  -159.451, Y  +684.743, Z    +0.000, E1   -38.666, E3 +130029.022}
SPL {X  -158.386, Y  +694.170, Z    +0.000, E1   -38.484, E3 +130055.140}
SPL {X  -157.286, Y  +700.846, Z    +0.000, E1   -38.194, E3 +130074.108}
SPL {X  -156.328, Y  +705.580, Z    +0.000, E1   -38.037, E3 +130087.644}
SPL {X  -155.162, Y  +710.549, Z    +0.000, E1   -37.822, E3 +130102.048}
SPL {X  -153.914, Y  +715.210, Z    +0.000, E1   -37.596, E3 +130115.697}
SPL {X  -152.686, Y  +719.322, Z    +0.000, E1   -37.361, E3 +130127.870}
SPL {X  -150.251, Y  +726.496, Z    +0.000, E1   -33.848, E3 +130176.365}
ENDSPLINE

SPLINE
SPL {X  -156.089, Y  +706.662, Z    +0.000, E1   -21.279, E3 +130229.019}
SPL {X  -159.059, Y  +688.824, Z    +0.000, E1   -11.551, E3 +130242.979}
SPL {X  -159.959, Y  +675.119, Z    +0.000, E1    -3.373, E3 +130247.807}
SPL {X  -160.000, Y  +666.447, Z    +0.000, E1    +3.005, E3 +130249.842}
SPL {X  -160.000, Y  +658.774, Z    +0.000, E1   +10.317, E3 +130252.101}
SPL {X  -160.000, Y  +647.765, Z    +0.000, E1   +20.359, E3 +130257.466}
SPL {X  -160.000, Y  +622.607, Z    +0.000, E1   +34.692, E3 +130280.333}
SPL {X  -160.000, Y  +596.106, Z    +0.000, E1   +39.718, E3 +130322.333}
SPL {X  -160.000, Y  +592.273, Z    +0.000, E1   +39.746, E3 +130332.071}
SPL {X  -160.000, Y  +586.287, Z    +0.000, E1   +39.762, E3 +130347.330}
SPL {X  -160.000, Y  +577.753, Z    +0.000, E1   +39.844, E3 +130368.972}
SPL {X  -160.000, Y  +567.367, Z    +0.000, E1   +39.853, E3 +130395.466}
SPL {X  -160.000, Y  +559.466, Z    +0.000, E1   +39.761, E3 +130415.747}
SPL {X  -160.000, Y  +552.914, Z    +0.000, E1   +39.787, E3 +130432.415}
SPL {X  -160.000, Y  +546.390, Z    +0.000, E1   +39.760, E3 +130449.128}
SPL {X  -160.000, Y  +540.123, Z    +0.000, E1   +39.770, E3 +130465.108}
SPL {X  -160.000, Y  +533.658, Z    +0.000, E1   +39.771, E3 +130481.606}
SPL {X  -160.000, Y  +527.046, Z    +0.000, E1   +39.771, E3 +130498.482}
SPL {X  -160.000, Y  +521.063, Z    +0.000, E1   +39.756, E3 +130513.766}
SPL {X  -160.000, Y  +515.110, Z    +0.000, E1   +39.770, E3 +130528.939}
SPL {X  -160.000, Y  +508.717, Z    +0.000, E1   +39.766, E3 +130545.257}
SPL {X  -160.000, Y  +502.133, Z    +0.000, E1   +39.780, E3 +130562.024}
ENDSPLINE

SPLINE
SPL {X  -160.000, Y  +512.949, Z    +0.000, E1   +32.050, E3 +130578.281}
ENDSPLINE

SPLINE
SPL {X  -160.000, Y  +507.092, Z    +0.000, E1   +32.805, E3 +130592.909}
SPL {X  -160.000, Y  +499.824, Z    +0.000, E1   +34.003, E3 +130608.651}
SPL {X  -160.000, Y  +491.367, Z    +0.000, E1   +35.449, E3 +130625.392}
SPL {X  -160.000, Y  +483.082, Z    +0.000, E1   +36.782, E3 +130641.231}
SPL {X  -160.000, Y  +474.521, Z    +0.000, E1   +38.037, E3 +130657.319}
SPL {X  -160.000, Y  +465.343, Z    +0.000, E1   +38.802, E3 +130677.477}
SPL {X  -160.000, Y  +457.266, Z    +0.000, E1   +38.756, E3 +130698.931}
SPL {X  -160.000, Y  +448.553, Z    +0.000, E1   +38.823, E3 +130721.882}
SPL {X  -160.000, Y  +439.425, Z    +0.000, E1   +38.797, E3 +130746.053}
SPL {X  -160.000, Y  +430.351, Z    +0.000, E1   +38.810, E3 +130770.068}
SPL {X  -160.000, Y  +421.477, Z    +0.000, E1   +38.792, E3 +130793.571}
SPL {X  -160.000, Y  +412.292, Z    +0.000, E1   +38.825, E3 +130817.799}
SPL {X  -160.000, Y  +403.281, Z    +0.000, E1   +38.797, E3 +130841.679}
SPL {X  -160.000, Y  +394.948, Z    +0.000, E1   +38.796, E3 +130863.721}
SPL {X  -159.971, Y  +385.741, Z    +0.000, E1   +38.831, E3 +130888.042}
SPL {X  -159.525, Y  +376.478, Z    +0.000, E1   +38.739, E3 +130913.033}
SPL {X  -158.721, Y  +368.613, Z    +0.000, E1   +38.561, E3 +130934.756}
SPL {X  -157.505, Y  +360.654, Z    +0.000, E1   +38.390, E3 +130957.029}
SPL {X  -156.229, Y  +354.269, Z    +0.000, E1   +38.076, E3 +130975.379}
SPL {X  -155.202, Y  +349.910, Z    +0.000, E1   +37.893, E3 +130987.953}
SPL {X  -154.128, Y  +345.852, Z    +0.000, E1   +37.701, E3 +130999.777}
SPL {X  -152.890, Y  +341.633, Z    +0.000, E1   +37.487, E3 +131012.209}
SPL {X  -150.284, Y  +333.893, Z    +0.000, E1   +33.433, E3 +131067.020}
ENDSPLINE

SPLINE
SPL {X  -157.404, Y  +360.095, Z    +0.000, E1   +17.695, E3 +131122.145}
SPL {X  -159.413, Y  +375.108, Z    +0.000, E1    +9.284, E3 +131131.233}
SPL {X  -159.978, Y  +386.135, Z    +0.000, E1    +2.544, E3 +131134.795}
SPL {X  -160.000, Y  +393.708, Z    +0.000, E1    -3.216, E3 +131136.548}
SPL {X  -160.000, Y  +400.474, Z    +0.000, E1    -9.529, E3 +131138.595}
SPL {X  -160.000, Y  +409.652, Z    +0.000, E1   -18.026, E3 +131142.731}
SPL {X  -160.000, Y  +437.804, Z    +0.000, E1   -34.779, E3 +131167.524}
SPL {X  -160.000, Y  +463.067, Z    +0.000, E1   -38.672, E3 +131213.224}
SPL {X  -160.000, Y  +469.167, Z    +0.000, E1   -38.717, E3 +131229.330}
SPL {X  -160.000, Y  +476.691, Z    +0.000, E1   -38.728, E3 +131249.262}
SPL {X  -160.000, Y  +483.419, Z    +0.000, E1   -38.692, E3 +131267.162}
SPL {X  -160.000, Y  +489.013, Z    +0.000, E1   -38.683, E3 +131282.001}
SPL {X  -160.000, Y  +494.786, Z    +0.000, E1   -38.693, E3 +131297.311}
SPL {X  -160.000, Y  +500.108, Z    +0.000, E1   -38.668, E3 +131311.462}
SPL {X  -160.000, Y  +504.903, Z    +0.000, E1   -38.673, E3 +131324.183}
SPL {X  -160.000, Y  +510.180, Z    +0.000, E1   -38.675, E3 +131338.188}
SPL {X  -160.000, Y  +515.083, Z    +0.000, E1   -38.662, E3 +131351.207}
SPL {X  -160.000, Y  +520.479, Z    +0.000, E1   -38.692, E3 +131365.482}
SPL {X  -160.000, Y  +525.998, Z    +0.000, E1   -38.666, E3 +131380.160}
SPL {X  -160.000, Y  +531.341, Z    +0.000, E1   -38.684, E3 +131394.304}
SPL {X  -160.000, Y  +537.313, Z    +0.000, E1   -38.686, E3 +131410.144}
SPL {X  -160.000, Y  +543.203, Z    +0.000, E1   -38.679, E3 +131425.770}
SPL {X  -160.000, Y  +551.201, Z    +0.000, E1   -38.768, E3 +131446.831}
SPL {X  -160.000, Y  +561.335, Z    +0.000, E1   -38.777, E3 +131473.701}
SPL {X  -160.000, Y  +568.812, Z    +0.000, E1   -38.671, E3 +131493.704}
SPL {X  -160.000, Y  +574.116, Z    +0.000, E1   -38.680, E3 +131507.775}
SPL {X  -160.000, Y  +582.193, Z    +0.000, E1   -38.759, E3 +131529.078}
SPL {X  -160.000, Y  +591.932, Z    +0.000, E1   -38.763, E3 +131554.903}
SPL {X  -160.000, Y  +601.488, Z    +0.000, E1   -38.747, E3 +131580.278}
SPL {X  -160.000, Y  +609.161, Z    +0.000, E1   -38.685, E3 +131600.730}
SPL {X  -160.000, Y  +614.445, Z    +0.000, E1   -38.661, E3 +131614.779}
SPL {X  -160.000, Y  +621.895, Z    +0.000, E1   -38.769, E3 +131634.368}
SPL {X  -160.000, Y  +631.692, Z    +0.000, E1   -38.748, E3 +131660.421}
SPL {X  -160.000, Y  +639.246, Z    +0.000, E1   -38.671, E3 +131680.597}
SPL {X  -160.000, Y  +644.827, Z    +0.000, E1   -38.662, E3 +131695.431}
SPL {X  -160.000, Y  +650.491, Z    +0.000, E1   -38.673, E3 +131710.419}
SPL {X  -160.000, Y  +656.011, Z    +0.000, E1   -38.669, E3 +131725.072}
SPL {X  -160.000, Y  +661.156, Z    +0.000, E1   -38.659, E3 +131738.747}
SPL {X  -160.000, Y  +666.701, Z    +0.000, E1   -38.683, E3 +131753.407}
SPL {X  -159.961, Y  +675.011, Z    +0.000, E1   -38.755, E3 +131775.394}
SPL {X  -159.451, Y  +684.743, Z    +0.000, E1   -38.666, E3 +131801.747}
SPL {X  -158.386, Y  +694.170, Z    +0.000, E1   -38.484, E3 +131827.866}
SPL {X  -157.286, Y  +700.846, Z    +0.000, E1   -38.194, E3 +131846.833}
SPL {X  -156.328, Y  +705.580, Z    +0.000, E1   -38.037, E3 +131860.369}
SPL {X  -155.162, Y  +710.549, Z    +0.000, E1   -37.822, E3 +131874.773}
SPL {X  -153.914, Y  +715.210, Z    +0.000, E1   -37.596, E3 +131888.423}
SPL {X  -152.686, Y  +719.322, Z    +0.000, E1   -37.361, E3 +131900.595}
SPL {X  -150.251, Y  +726.496, Z    +0.000, E1   -33.848, E3 +131949.091}
ENDSPLINE

SPLINE
SPL {X  -156.089, Y  +706.662, Z    +0.000, E1   -21.279, E3 +132001.744}
SPL {X  -159.059, Y  +688.824, Z    +0.000, E1   -11.551, E3 +132015.704}
SPL {X  -159.959, Y  +675.119, Z    +0.000, E1    -3.373, E3 +132020.533}
SPL {X  -160.000, Y  +666.447, Z    +0.000, E1    +3.005, E3 +132022.567}
SPL {X  -160.000, Y  +658.774, Z    +0.000, E1   +10.317, E3 +132024.826}
SPL {X  -160.000, Y  +647.765, Z    +0.000, E1   +20.359, E3 +132030.191}
SPL {X  -160.000, Y  +622.607, Z    +0.000, E1   +34.692, E3 +132053.058}
SPL {X  -160.000, Y  +596.106, Z    +0.000, E1   +39.718, E3 +132095.058}
SPL {X  -160.000, Y  +592.273, Z    +0.000, E1   +39.746, E3 +132104.796}
SPL {X  -160.000, Y  +586.287, Z    +0.000, E1   +39.762, E3 +132120.055}
SPL {X  -160.000, Y  +577.753, Z    +0.000, E1   +39.844, E3 +132141.697}
SPL {X  -160.000, Y  +567.367, Z    +0.000, E1   +39.853, E3 +132168.191}
SPL {X  -160.000, Y  +559.466, Z    +0.000, E1   +39.761, E3 +132188.472}
SPL {X  -160.000, Y  +552.914, Z    +0.000, E1   +39.787, E3 +132205.140}
SPL {X  -160.000, Y  +546.390, Z    +0.000, E1   +39.760, E3 +132221.854}
SPL {X  -160.000, Y  +540.123, Z    +0.000, E1   +39.770, E3 +132237.833}
SPL {X  -160.000, Y  +533.658, Z    +0.000, E1   +39.771, E3 +132254.331}
SPL {X  -160.000, Y  +527.046, Z    +0.000, E1   +39.771, E3 +132271.207}
SPL {X  -160.000, Y  +521.063, Z    +0.000, E1   +39.756, E3 +132286.492}
SPL {X  -160.000, Y  +515.110, Z    +0.000, E1   +39.770, E3 +132301.664}
SPL {X  -160.000, Y  +508.717, Z    +0.000, E1   +39.766, E3 +132317.983}
SPL {X  -160.000, Y  +502.133, Z    +0.000, E1   +39.780, E3 +132334.749}
ENDSPLINE

SPLINE
SPL {X  -160.000, Y  +512.949, Z    +0.000, E1   +32.050, E3 +132351.006}
ENDSPLINE

SPLINE
SPL {X  -160.000, Y  +507.092, Z    +0.000, E1   +32.805, E3 +132365.635}
SPL {X  -160.000, Y  +499.824, Z    +0.000, E1   +34.003, E3 +132381.376}
SPL {X  -160.000, Y  +491.367, Z    +0.000, E1   +35.449, E3 +132398.117}
SPL {X  -160.000, Y  +483.082, Z    +0.000, E1   +36.782, E3 +132413.956}
SPL {X  -160.000, Y  +474.521, Z    +0.000, E1   +38.037, E3 +132430.044}
SPL {X  -160.000, Y  +465.343, Z    +0.000, E1   +38.802, E3 +132450.203}
SPL {X  -160.000, Y  +457.266, Z    +0.000, E1   +38.756, E3 +132471.656}
SPL {X  -160.000, Y  +448.553, Z    +0.000, E1   +38.823, E3 +132494.607}
SPL {X  -160.000, Y  +439.425, Z    +0.000, E1   +38.797, E3 +132518.778}
SPL {X  -160.000, Y  +430.351, Z    +0.000, E1   +38.810, E3 +132542.793}
SPL {X  -160.000, Y  +421.477, Z    +0.000, E1   +38.792, E3 +132566.297}
SPL {X  -160.000, Y  +412.292, Z    +0.000, E1   +38.825, E3 +132590.524}
SPL {X  -160.000, Y  +403.281, Z    +0.000, E1   +38.797, E3 +132614.404}
SPL {X  -160.000, Y  +394.948, Z    +0.000, E1   +38.796, E3 +132636.446}
SPL {X  -159.971, Y  +385.741, Z    +0.000, E1   +38.831, E3 +132660.767}
SPL {X  -159.525, Y  +376.478, Z    +0.000, E1   +38.739, E3 +132685.758}
SPL {X  -158.721, Y  +368.613, Z    +0.000, E1   +38.561, E3 +132707.481}
SPL {X  -157.505, Y  +360.654, Z    +0.000, E1   +38.390, E3 +132729.754}
SPL {X  -156.229, Y  +354.269, Z    +0.000, E1   +38.076, E3 +132748.104}
SPL {X  -155.202, Y  +349.910, Z    +0.000, E1   +37.893, E3 +132760.679}
SPL {X  -154.128, Y  +345.852, Z    +0.000, E1   +37.701, E3 +132772.503}
SPL {X  -152.890, Y  +341.633, Z    +0.000, E1   +37.487, E3 +132784.935}
SPL {X  -150.284, Y  +333.893, Z    +0.000, E1   +33.433, E3 +132839.745}
ENDSPLINE

SPLINE
SPL {X  -157.404, Y  +360.095, Z    +0.000, E1   +17.695, E3 +132894.870}
SPL {X  -159.413, Y  +375.108, Z    +0.000, E1    +9.284, E3 +132903.959}
SPL {X  -159.978, Y  +386.135, Z    +0.000, E1    +2.544, E3 +132907.520}
SPL {X  -160.000, Y  +393.708, Z    +0.000, E1    -3.216, E3 +132909.274}
SPL {X  -160.000, Y  +400.474, Z    +0.000, E1    -9.529, E3 +132911.320}
SPL {X  -160.000, Y  +409.652, Z    +0.000, E1   -18.026, E3 +132915.457}
SPL {X  -160.000, Y  +437.804, Z    +0.000, E1   -34.779, E3 +132940.249}
SPL {X  -160.000, Y  +463.067, Z    +0.000, E1   -38.672, E3 +132985.949}
SPL {X  -160.000, Y  +469.167, Z    +0.000, E1   -38.717, E3 +133002.056}
SPL {X  -160.000, Y  +476.691, Z    +0.000, E1   -38.728, E3 +133021.987}
SPL {X  -160.000, Y  +483.419, Z    +0.000, E1   -38.692, E3 +133039.887}
SPL {X  -160.000, Y  +489.013, Z    +0.000, E1   -38.683, E3 +133054.726}
SPL {X  -160.000, Y  +494.786, Z    +0.000, E1   -38.693, E3 +133070.036}
SPL {X  -160.000, Y  +500.108, Z    +0.000, E1   -38.668, E3 +133084.188}
SPL {X  -160.000, Y  +504.903, Z    +0.000, E1   -38.673, E3 +133096.909}
SPL {X  -160.000, Y  +510.180, Z    +0.000, E1   -38.675, E3 +133110.913}
SPL {X  -160.000, Y  +515.083, Z    +0.000, E1   -38.662, E3 +133123.933}
SPL {X  -160.000, Y  +520.479, Z    +0.000, E1   -38.692, E3 +133138.207}
SPL {X  -160.000, Y  +525.998, Z    +0.000, E1   -38.666, E3 +133152.885}
SPL {X  -160.000, Y  +531.341, Z    +0.000, E1   -38.684, E3 +133167.029}
SPL {X  -160.000, Y  +537.313, Z    +0.000, E1   -38.686, E3 +133182.869}
SPL {X  -160.000, Y  +543.203, Z    +0.000, E1   -38.679, E3 +133198.495}
SPL {X  -160.000, Y  +551.201, Z    +0.000, E1   -38.768, E3 +133219.556}
SPL {X  -160.000, Y  +561.335, Z    +0.000, E1   -38.777, E3 +133246.426}
SPL {X  -160.000, Y  +568.812, Z    +0.000, E1   -38.671, E3 +133266.430}
SPL {X  -160.000, Y  +574.116, Z    +0.000, E1   -38.680, E3 +133280.500}
SPL {X  -160.000, Y  +582.193, Z    +0.000, E1   -38.759, E3 +133301.804}
SPL {X  -160.000, Y  +591.932, Z    +0.000, E1   -38.763, E3 +133327.629}
SPL {X  -160.000, Y  +601.488, Z    +0.000, E1   -38.747, E3 +133353.004}
SPL {X  -160.000, Y  +609.161, Z    +0.000, E1   -38.685, E3 +133373.456}
SPL {X  -160.000, Y  +614.445, Z    +0.000, E1   -38.661, E3 +133387.505}
SPL {X  -160.000, Y  +621.895, Z    +0.000, E1   -38.769, E3 +133407.093}
SPL {X  -160.000, Y  +631.692, Z    +0.000, E1   -38.748, E3 +133433.146}
SPL {X  -160.000, Y  +639.246, Z    +0.000, E1   -38.671, E3 +133453.322}
SPL {X  -160.000, Y  +644.827, Z    +0.000, E1   -38.662, E3 +133468.157}
SPL {X  -160.000, Y  +650.491, Z    +0.000, E1   -38.673, E3 +133483.144}
SPL {X  -160.000, Y  +656.011, Z    +0.000, E1   -38.669, E3 +133497.797}
SPL {X  -160.000, Y  +661.156, Z    +0.000, E1   -38.659, E3 +133511.472}
SPL {X  -160.000, Y  +666.701, Z    +0.000, E1   -38.683, E3 +133526.132}
SPL {X  -159.961, Y  +675.011, Z    +0.000, E1   -38.755, E3 +133548.119}
SPL {X  -159.451, Y  +684.743, Z    +0.000, E1   -38.666, E3 +133574.472}
SPL {X  -158.386, Y  +694.170, Z    +0.000, E1   -38.484, E3 +133600.591}
SPL {X  -157.286, Y  +700.846, Z    +0.000, E1   -38.194, E3 +133619.559}
SPL {X  -156.328, Y  +705.580, Z    +0.000, E1   -38.037, E3 +133633.095}
SPL {X  -155.162, Y  +710.549, Z    +0.000, E1   -37.822, E3 +133647.498}
SPL {X  -153.914, Y  +715.210, Z    +0.000, E1   -37.596, E3 +133661.148}
SPL {X  -152.686, Y  +719.322, Z    +0.000, E1   -37.361, E3 +133673.320}
SPL {X  -150.251, Y  +726.496, Z    +0.000, E1   -33.848, E3 +133721.816}
ENDSPLINE

SPLINE
SPL {X  -156.089, Y  +706.662, Z    +0.000, E1   -21.279, E3 +133774.469}
SPL {X  -159.059, Y  +688.824, Z    +0.000, E1   -11.551, E3 +133788.430}
SPL {X  -159.959, Y  +675.119, Z    +0.000, E1    -3.373, E3 +133793.258}
SPL {X  -160.000, Y  +666.447, Z    +0.000, E1    +3.005, E3 +133795.293}
SPL {X  -160.000, Y  +658.774, Z    +0.000, E1   +10.317, E3 +133797.551}
SPL {X  -160.000, Y  +647.765, Z    +0.000, E1   +20.359, E3 +133802.916}
SPL {X  -160.000, Y  +622.607, Z    +0.000, E1   +34.692, E3 +133825.784}
SPL {X  -160.000, Y  +596.106, Z    +0.000, E1   +39.718, E3 +133867.784}
SPL {X  -160.000, Y  +592.273, Z    +0.000, E1   +39.746, E3 +133877.521}
SPL {X  -160.000, Y  +586.287, Z    +0.000, E1   +39.762, E3 +133892.780}
SPL {X  -160.000, Y  +577.753, Z    +0.000, E1   +39.844, E3 +133914.422}
SPL {X  -160.000, Y  +567.367, Z    +0.000, E1   +39.853, E3 +133940.916}
SPL {X  -160.000, Y  +559.466, Z    +0.000, E1   +39.761, E3 +133961.198}
SPL {X  -160.000, Y  +552.914, Z    +0.000, E1   +39.787, E3 +133977.865}
SPL {X  -160.000, Y  +546.390, Z    +0.000, E1   +39.760, E3 +133994.579}
SPL {X  -160.000, Y  +540.123, Z    +0.000, E1   +39.770, E3 +134010.558}
SPL {X  -160.000, Y  +533.658, Z    +0.000, E1   +39.771, E3 +134027.057}
SPL {X  -160.000, Y  +527.046, Z    +0.000, E1   +39.771, E3 +134043.932}
SPL {X  -160.000, Y  +521.063, Z    +0.000, E1   +39.756, E3 +134059.217}
SPL {X  -160.000, Y  +515.110, Z    +0.000, E1   +39.770, E3 +134074.389}
SPL {X  -160.000, Y  +508.717, Z    +0.000, E1   +39.766, E3 +134090.708}
SPL {X  -160.000, Y  +502.133, Z    +0.000, E1   +39.780, E3 +134107.474}
ENDSPLINE

SPLINE
SPL {X  -160.000, Y  +512.949, Z    +0.000, E1   +32.050, E3 +134123.732}
ENDSPLINE

SPLINE
SPL {X  -160.000, Y  +507.092, Z    +0.000, E1   +32.805, E3 +134138.360}
SPL {X  -160.000, Y  +499.824, Z    +0.000, E1   +34.003, E3 +134154.102}
SPL {X  -160.000, Y  +491.367, Z    +0.000, E1   +35.449, E3 +134170.842}
SPL {X  -160.000, Y  +483.082, Z    +0.000, E1   +36.782, E3 +134186.681}
SPL {X  -160.000, Y  +474.521, Z    +0.000, E1   +38.037, E3 +134202.769}
SPL {X  -160.000, Y  +465.343, Z    +0.000, E1   +38.802, E3 +134222.928}
SPL {X  -160.000, Y  +457.266, Z    +0.000, E1   +38.756, E3 +134244.382}
SPL {X  -160.000, Y  +448.553, Z    +0.000, E1   +38.823, E3 +134267.333}
SPL {X  -160.000, Y  +439.425, Z    +0.000, E1   +38.797, E3 +134291.504}
SPL {X  -160.000, Y  +430.351, Z    +0.000, E1   +38.810, E3 +134315.518}
SPL {X  -160.000, Y  +421.477, Z    +0.000, E1   +38.792, E3 +134339.022}
SPL {X  -160.000, Y  +412.292, Z    +0.000, E1   +38.825, E3 +134363.249}
SPL {X  -160.000, Y  +403.281, Z    +0.000, E1   +38.797, E3 +134387.129}
SPL {X  -160.000, Y  +394.948, Z    +0.000, E1   +38.796, E3 +134409.171}
SPL {X  -159.971, Y  +385.741, Z    +0.000, E1   +38.831, E3 +134433.492}
SPL {X  -159.525, Y  +376.478, Z    +0.000, E1   +38.739, E3 +134458.483}
SPL {X  -158.721, Y  +368.613, Z    +0.000, E1   +38.561, E3 +134480.206}
SPL {X  -157.505, Y  +360.654, Z    +0.000, E1   +38.390, E3 +134502.480}
SPL {X  -156.229, Y  +354.269, Z    +0.000, E1   +38.076, E3 +134520.829}
SPL {X  -155.202, Y  +349.910, Z    +0.000, E1   +37.893, E3 +134533.404}
SPL {X  -154.128, Y  +345.852, Z    +0.000, E1   +37.701, E3 +134545.228}
SPL {X  -152.890, Y  +341.633, Z    +0.000, E1   +37.487, E3 +134557.660}
SPL {X  -150.284, Y  +333.893, Z    +0.000, E1   +33.433, E3 +134612.470}
ENDSPLINE

